// TwinCAT 3 PLC project Test
// ProgramVersion: 3.1.4026.24
// libraries:
//   Tc2_Standard, * (Beckhoff Automation GmbH)
//   Tc2_System, * (Beckhoff Automation GmbH)
// project tree:
//   DUTs/AMR/ stJoint2.TcDUT, stPose2D.TcDUT, stTarget2D.TcDUT
//   DUTs/BaseActions/ ITF_BA_6Axis.TcIO, ITF_BA_AMR.TcIO, ITF_BA_Scara.TcIO
//   DUTs/BasicRobot/ eMode.TcDUT, stFrame.TcDUT, stPose.TcDUT, stTarget.TcDUT
//   DUTs/Communication/ eCommunicationState.TcDUT, ITF_CommunicationModul_1.TcIO, ST_CommunicationConfig_1.TcDUT
//   DUTs/DB/ ST_Robot.TcDUT, ST_SQLValue.TcDUT
//   DUTs/Error/ eSeverity.TcDUT, stError.TcDUT
//   DUTs/ ITF_0_BaseComponent.TcIO, ITF_1_Robot.TcIO, ITF_1_Skill.TcIO, ITF_2_6AxisRobot.TcIO, ITF_2_AMR.TcIO, ITF_CommunicationModul.TcIO, ITF_Tool.TcIO, ST_CommunicationConfig.TcDUT
//   DUTs/Manipulator/ ITF_Tool_1.TcIO, stJoint6.TcDUT, stPose3D.TcDUT, stTarget3D.TcDUT
//   DUTs/StateMachine/ eInternalTransitions.TcDUT, eResult.TcDUT, eState.TcDUT, eSupervisoryTransitions.TcDUT
//   GVLs/ OPCUA.TcGVL, SKILLS.TcGVL
//   / PlcTask.TcTTO
//   POUs/Archiv/ FB_Axis.TcPOU
//   POUs/ FB_Base.TcPOU, FB_Helper.TcPOU, FB_PickPlaceSkill.TcPOU, FB_PostgreSQLClient.TcPOU, FB_ROB.TcPOU, FB_ROB_AMR.TcPOU, FB_ROB_MANIP.TcPOU, FB_Skill.TcPOU, FB_SkillHandler.TcPOU, FB_Tool.TcPOU, FB_UR5.TcPOU, MAIN_1.TcPOU, Test.TcPOU
//   POUs/Robots/ FB_OmronLD90.TcPOU, FB_ROB_1.TcPOU, FB_ROB_AMR_1.TcPOU, FB_ROB_MANIP_1.TcPOU, FB_UR5_1.TcPOU
//   POUs/Skills/ FB_SkillHandler_1.TcPOU, FB_Skill_1.TcPOU, Skill_LoadDeliverReturn.TcPOU, Skill_PickPlace.TcPOU

CONFIGURATION Test
    RESOURCE PLC ON TwinCAT3
        TASK PlcTask(INTERVAL := T#10ms, PRIORITY := 21);
        PROGRAM MAIN WITH PlcTask : MAIN;
    END_RESOURCE
END_CONFIGURATION

// ---- DUTs/AMR/stJoint2.TcDUT
TYPE stJoint2 :
STRUCT
	left : LREAL;
	right : LREAL;
END_STRUCT
END_TYPE

// ---- DUTs/AMR/stPose2D.TcDUT
TYPE stPose2D EXTENDS stPose :
STRUCT
	theta : LREAL;
END_STRUCT
END_TYPE

// ---- DUTs/AMR/stTarget2D.TcDUT
TYPE stTarget2D EXTENDS stTarget :
STRUCT
	pose : stPose2D;
END_STRUCT
END_TYPE

// ---- DUTs/BasicRobot/eMode.TcDUT
{attribute 'qualified_only'}
{attribute 'strict'}
TYPE eMode :
(
	Manual := 0,
	Automatic := 1
);
END_TYPE

// ---- DUTs/BasicRobot/stFrame.TcDUT
TYPE stFrame :
STRUCT
	frameId: UINT;
END_STRUCT
END_TYPE

// ---- DUTs/BasicRobot/stPose.TcDUT
TYPE stPose :
STRUCT
	x : LREAL;
	y : LREAL;
END_STRUCT
END_TYPE

// ---- DUTs/BasicRobot/stTarget.TcDUT
TYPE stTarget :
STRUCT
	name : STRING(80);
	frameId : INT;
END_STRUCT
END_TYPE

// ---- DUTs/Communication/eCommunicationState.TcDUT
{attribute 'qualified_only'}
{attribute 'strict'}
{attribute 'to_string'}
TYPE eCommunicationState :
(
	DISCONNECTED,
    CONNECTING,
    CONNECTED,
    DISCONNECTING,
    ERROR
);
END_TYPE

// ---- DUTs/Communication/ST_CommunicationConfig_1.TcDUT
TYPE ST_CommunicationConfig_1 :
STRUCT

    sIpAddress : STRING(15) := '192.168.0.10';
    nPort : UINT := 7171;
	sUsername: STRING(128):= '';
    sPassword : STRING(128) := '';
    tTimeout : TIME := T#5S;
    bAutoReconnect : BOOL := TRUE;
END_STRUCT
END_TYPE

// ---- DUTs/DB/ST_Robot.TcDUT
TYPE ST_Robot :
STRUCT
    id           : DINT;
    name         : STRING(80);
    manufacturer : STRING(80);
    model        : STRING(80);
    robot_type   : STRING(80);
    axes         : DINT;
    payload      : LREAL;
    reach        : LREAL;
    controller   : STRING(80);
    ip_address   : STRING(40);
END_STRUCT
END_TYPE

// ---- DUTs/DB/ST_SQLValue.TcDUT
TYPE ST_SQLValue  :
STRUCT
    sValue : STRING(255);
END_STRUCT
END_TYPE

// ---- DUTs/Error/eSeverity.TcDUT
{attribute 'qualified_only'}
{attribute 'strict'}
TYPE eSeverity :
(
	Info := 0,
	Warning := 1,
	Error := 2,
	Critical := 3
);
END_TYPE

// ---- DUTs/Error/stError.TcDUT
TYPE stError :
STRUCT
	code : INT;
	message : STRING(255);
	timestamp : DATE_AND_TIME;
	severity : eSeverity;
END_STRUCT
END_TYPE

// ---- DUTs/Manipulator/stJoint6.TcDUT
TYPE stJoint6 :
STRUCT
	joint1 : LREAL;
	joint2 : LREAL;
	joint3 : LREAL;
	joint4 : LREAL;
	joint5 : LREAL;
	joint6 : LREAL;
END_STRUCT
END_TYPE

// ---- DUTs/Manipulator/stPose3D.TcDUT
TYPE stPose3D EXTENDS stPose :
STRUCT
	z : LREAL;
	rx : LREAL;
	ry : LREAL;
	rz : LREAL;
END_STRUCT
END_TYPE

// ---- DUTs/Manipulator/stTarget3D.TcDUT
TYPE stTarget3D EXTENDS stTarget :
STRUCT
	pose : stPose3D;
END_STRUCT
END_TYPE

// ---- DUTs/StateMachine/eInternalTransitions.TcDUT
{attribute 'qualified_only'}
{attribute 'strict'}
TYPE eInternalTransitions :
(
	Configuring := 0,
	CleaningUp := 1,
	ShuttingDown := 2,
	Activating := 3,
	Deactivating := 4,
	ErrorProcessing := 5
);
END_TYPE

// ---- DUTs/StateMachine/eResult.TcDUT
{attribute 'qualified_only'}
{attribute 'strict'}
{attribute 'to_string'}
TYPE eResult :
(
	NONE := 0,
	SUCCESS := 1,
	FAILURE := 2,
	ERROR	:= 3
);
END_TYPE

// ---- DUTs/StateMachine/eState.TcDUT
{attribute 'qualified_only'}
{attribute 'strict'}
TYPE eState :
(
	None 			:= 0,
	Unconfigured 	:= 1,
	Inactive 		:= 2,
	Active 			:= 3,
	Finalized 		:= 4,
	Configuring		:= 5,
	CleaningUp 		:= 6,
	Activating 		:= 7,
	Deactivating 	:= 8,
	ShuttingDown 	:= 9,
	ErrorProcessing := 10
);
END_TYPE

// ---- DUTs/StateMachine/eSupervisoryTransitions.TcDUT
{attribute 'qualified_only'}
{attribute 'strict'}
TYPE eSupervisoryTransitions :
(
	create := 0,
	configure := 1,
	cleanup := 2,
	activate := 3,
	deactivate := 4,
	shutdown := 5,
	destroy := 6
);
END_TYPE

// ---- DUTs/ST_CommunicationConfig.TcDUT
TYPE ST_CommunicationConfig :
STRUCT
	sIPAdress: STRING;
	Port: UINT;
	
END_STRUCT
END_TYPE

// ---- GVLs/OPCUA.TcGVL
{attribute 'qualified_only'}
VAR_GLOBAL
	{attribute 'OPC.UA.DA.StructuredType' := '1'}
	{attribute 'OPC.UA.DA' := '1'}
	ROB : ARRAY[1..3] of FB_ROB;
END_VAR

// ---- GVLs/SKILLS.TcGVL
{attribute 'qualified_only'}
VAR_GLOBAL
	PnP: FB_PickPlaceSkill;
END_VAR

// ---- DUTs/BaseActions/ITF_BA_6Axis.TcIO
INTERFACE ITF_BA_6Axis

METHOD MC_ChangeSpeedOverride : INT
VAR_INPUT
	factor: REAL;
END_VAR
END_METHOD

METHOD MC_MoveAxesAbsolute : BOOL
VAR_INPUT
	target: stTarget3D;
END_VAR
END_METHOD

METHOD MC_MoveAxesRelative : BOOL
VAR_INPUT
	axes: ARRAY[1..6] OF FB_Axis;
	offsets: ARRAY[1..6] OF REAL;
END_VAR
END_METHOD

METHOD MC_MoveLinearAbsolute : BOOL
VAR_INPUT
	target: stTarget3D;
END_VAR
END_METHOD

METHOD PUBLIC MC_ReadAnalogInput : LREAL
VAR_INPUT
	input : INT;
END_VAR
END_METHOD

METHOD PUBLIC MC_ReadDigitalInput : BOOL
VAR_INPUT
	input : INT;
END_VAR
END_METHOD

METHOD PUBLIC MC_SetDigitalOutput : BOOL
VAR_INPUT
	output : INT;
	value : BOOL;
END_VAR
END_METHOD

METHOD PUBLIC MC_SetOperationMode : BOOL
VAR_INPUT
	mode: eMode;
END_VAR
END_METHOD

END_INTERFACE

// ---- DUTs/BaseActions/ITF_BA_AMR.TcIO
INTERFACE ITF_BA_AMR

METHOD MC_ChangeSpeedOverride : INT
VAR_INPUT
	factor: REAL;
END_VAR
END_METHOD

METHOD MC_MoveAxesAbsolute : BOOL
VAR_INPUT
	target: stTarget3D;
END_VAR
END_METHOD

METHOD MC_MoveAxesRelative : BOOL
VAR_INPUT
	axes: ARRAY[1..6] OF FB_Axis;
	offsets: ARRAY[1..6] OF REAL;
END_VAR
END_METHOD

METHOD MC_MoveLinearAbsolute : BOOL
VAR_INPUT
	target: stTarget3D;
END_VAR
END_METHOD

METHOD PUBLIC MC_ReadAnalogInput : LREAL
VAR_INPUT
	input : INT;
END_VAR
END_METHOD

METHOD PUBLIC MC_ReadDigitalInput : BOOL
VAR_INPUT
	input : INT;
END_VAR
END_METHOD

METHOD PUBLIC MC_SetDigitalOutput : BOOL
VAR_INPUT
	output : INT;
	value : BOOL;
END_VAR
END_METHOD

METHOD PUBLIC MC_SetOperationMode : BOOL
VAR_INPUT
	mode: eMode;
END_VAR
END_METHOD

END_INTERFACE

// ---- DUTs/BaseActions/ITF_BA_Scara.TcIO
INTERFACE ITF_BA_Scara

METHOD MC_ChangeSpeedOverride : INT
VAR_INPUT
	factor: REAL;
END_VAR
END_METHOD

METHOD MC_MoveAxesAbsolute : BOOL
VAR_INPUT
	target: stTarget3D;
END_VAR
END_METHOD

METHOD MC_MoveAxesRelative : BOOL
VAR_INPUT
	axes: ARRAY[1..6] OF FB_Axis;
	offsets: ARRAY[1..6] OF REAL;
END_VAR
END_METHOD

METHOD MC_MoveLinearAbsolute : BOOL
VAR_INPUT
	target: stTarget3D;
END_VAR
END_METHOD

METHOD PUBLIC MC_ReadAnalogInput : LREAL
VAR_INPUT
	input : INT;
END_VAR
END_METHOD

METHOD PUBLIC MC_ReadDigitalInput : BOOL
VAR_INPUT
	input : INT;
END_VAR
END_METHOD

METHOD PUBLIC MC_SetDigitalOutput : BOOL
VAR_INPUT
	output : INT;
	value : BOOL;
END_VAR
END_METHOD

METHOD PUBLIC MC_SetOperationMode : BOOL
VAR_INPUT
	mode: eMode;
END_VAR
END_METHOD

END_INTERFACE

// ---- DUTs/Communication/ITF_CommunicationModul_1.TcIO
INTERFACE ITF_CommunicationModul_1

METHOD Connect : BOOL
VAR_INPUT
END_VAR
END_METHOD

PROPERTY Connected : BOOL
GET
END_GET
END_PROPERTY

METHOD Disconnect : BOOL
VAR_INPUT
END_VAR
END_METHOD

METHOD ResetConnection : BOOL
VAR_INPUT
END_VAR
END_METHOD

END_INTERFACE

// ---- DUTs/ITF_0_BaseComponent.TcIO
INTERFACE ITF_0_BaseComponent

METHOD M_activate : BOOL
VAR_INPUT
END_VAR
END_METHOD

METHOD M_cleanup : BOOL
VAR_INPUT
END_VAR
END_METHOD

METHOD M_configure : BOOL
VAR_INPUT
END_VAR
END_METHOD

METHOD M_deactivate : BOOL
VAR_INPUT
END_VAR
END_METHOD

METHOD M_destroy : BOOL
VAR_INPUT
END_VAR
END_METHOD

METHOD M_shutdown : BOOL
VAR_INPUT
END_VAR
END_METHOD

METHOD onActivate : BOOL
VAR_INPUT
END_VAR
END_METHOD

METHOD onCleanup : BOOL
VAR_INPUT
END_VAR
END_METHOD

METHOD onConfigure : BOOL
VAR_INPUT
END_VAR
END_METHOD

METHOD onDeactivate : BOOL
VAR_INPUT
END_VAR
END_METHOD

METHOD onError : BOOL
VAR_INPUT
END_VAR
END_METHOD

METHOD onShutdown : BOOL
VAR_INPUT
END_VAR
END_METHOD

PROPERTY P_ID : UINT
GET
END_GET
SET
END_SET
END_PROPERTY

PROPERTY P_Name : String
GET
END_GET
END_PROPERTY

PROPERTY P_Path : String
GET
END_GET
END_PROPERTY

PROPERTY ABSTRACT P_State : eState
GET
END_GET
SET
END_SET
END_PROPERTY

END_INTERFACE

// ---- DUTs/ITF_1_Robot.TcIO
INTERFACE ITF_1_Robot EXTENDS ITF_0_BaseComponent

METHOD M_AUTO : BOOL
VAR_INPUT
END_VAR
END_METHOD

METHOD M_Disable : BOOL
VAR_INPUT
END_VAR
END_METHOD

METHOD M_DisableVelocityOverride : BOOL
VAR_INPUT
END_VAR
END_METHOD

METHOD M_Enable : BOOL
VAR_INPUT
END_VAR
END_METHOD

METHOD M_EnableVelocityOverride : BOOL
VAR_INPUT
END_VAR
END_METHOD

METHOD M_EStop : BOOL
VAR_INPUT
END_VAR
END_METHOD

METHOD M_MAN : BOOL
VAR_INPUT
END_VAR
END_METHOD

PROPERTY P_isInCollision : BOOL
GET
END_GET
END_PROPERTY

{warning 'Eigenschaftenimplementierung hinzufügen'}
PROPERTY P_JogSpeed : LREAL
GET
END_GET
SET
END_SET
END_PROPERTY

{warning 'Eigenschaftenimplementierung hinzufügen'}
PROPERTY P_RobotIsMoving : BOOL
GET
END_GET
END_PROPERTY

{warning 'Eigenschaftenimplementierung hinzufügen'}
PROPERTY P_RobotIsReady : BOOL
GET
END_GET
END_PROPERTY

END_INTERFACE

// ---- DUTs/ITF_1_Skill.TcIO
INTERFACE ITF_1_Skill EXTENDS ITF_0_BaseComponent

METHOD M_Pause : BOOL
VAR_INPUT
END_VAR
END_METHOD

METHOD M_Restart : BOOL
VAR_INPUT
END_VAR
END_METHOD

METHOD M_Resume : BOOL
VAR_INPUT
END_VAR
END_METHOD

METHOD M_Start : BOOL
VAR_INPUT
END_VAR
END_METHOD

METHOD M_Stop : BOOL
VAR_INPUT
END_VAR
END_METHOD

PROPERTY P_Busy : BOOL
GET
END_GET
END_PROPERTY

PROPERTY P_Done : BOOL
GET
END_GET
END_PROPERTY

END_INTERFACE

// ---- DUTs/ITF_2_6AxisRobot.TcIO
INTERFACE ITF_2_6AxisRobot IMPLEMENTS ITF_1_Robot

METHOD M_Home : BOOL
VAR_INPUT
END_VAR
END_METHOD

METHOD M_SwitchTool : UINT
VAR_INPUT
	tool: FB_Tool;
END_VAR
END_METHOD

{warning 'Eigenschaftenimplementierung hinzufügen'}
PROPERTY P_ActualAxisPos :stJoint6
GET
END_GET
END_PROPERTY

PROPERTY P_ActualJointVelocity : stJoint6
GET
END_GET
END_PROPERTY

{warning 'Eigenschaftenimplementierung hinzufügen'}
PROPERTY P_ActualTCPPos :stPose3D
GET
END_GET
END_PROPERTY

PROPERTY P_ActualTCPVelocity : stPose3D
GET
END_GET
END_PROPERTY

PROPERTY P_CurrentFrame : stFrame
GET
END_GET
SET
END_SET
END_PROPERTY

PROPERTY P_CurrentFrameID : UINT
GET
END_GET
END_PROPERTY

PROPERTY P_CurrentTool : FB_Tool
GET
END_GET
SET
END_SET
END_PROPERTY

PROPERTY P_IsInHomePosition : BOOL
GET
END_GET
END_PROPERTY

{warning 'Add property implementation'}
PROPERTY P_TargetReached : BOOL
GET
END_GET
END_PROPERTY

END_INTERFACE

// ---- DUTs/ITF_2_AMR.TcIO
INTERFACE ITF_2_AMR IMPLEMENTS ITF_1_Robot

METHOD M_Dock : BOOL
VAR_INPUT
END_VAR
END_METHOD

PROPERTY P_ActualAxisPos :stJoint2
GET
END_GET
END_PROPERTY

PROPERTY P_ActualJointVelocity : stJoint2
GET
END_GET
END_PROPERTY

PROPERTY P_ActualTCPPos :stPose2D
GET
END_GET
END_PROPERTY

PROPERTY P_ActualTCPVelocity : stPose2D
GET
END_GET
END_PROPERTY

PROPERTY P_IsDocked : BOOL
GET
END_GET
END_PROPERTY

{warning 'Add property implementation'}
PROPERTY P_TargetReached : BOOL
GET
END_GET
END_PROPERTY

END_INTERFACE

// ---- DUTs/ITF_CommunicationModul.TcIO
INTERFACE ITF_CommunicationModul

METHOD M_Connect : BOOL
VAR_INPUT
END_VAR
END_METHOD

METHOD M_Disconnect : BOOL
VAR_INPUT
END_VAR
END_METHOD

METHOD M_ResetConnection : BOOL
VAR_INPUT
END_VAR
END_METHOD

PROPERTY P_bConnected : BOOL
GET
END_GET
END_PROPERTY

END_INTERFACE

// ---- DUTs/ITF_Tool.TcIO
INTERFACE ITF_Tool

METHOD Grip : BOOL
VAR_INPUT
END_VAR
END_METHOD

METHOD Release : BOOL
VAR_INPUT
END_VAR
END_METHOD

END_INTERFACE

// ---- DUTs/Manipulator/ITF_Tool_1.TcIO
INTERFACE ITF_Tool_1

METHOD Grip : BOOL
VAR_INPUT
END_VAR
END_METHOD

METHOD Release : BOOL
VAR_INPUT
END_VAR
END_METHOD

END_INTERFACE

// ---- POUs/FB_ROB.TcPOU
FUNCTION_BLOCK FB_ROB EXTENDS FB_Base IMPLEMENTS ITF_1_Robot

// VAR_IN_OUT
// 	Skills: ARRAY[1..3] OF FB_Skill;
// END_VAR
VAR_INPUT
	ComConfig: ST_CommunicationConfig;
END_VAR


VAR_OUTPUT
	_inCollision: BOOL;
END_VAR
VAR
	_enabled: BOOL;
	_mode: eMode;
	_locked: BOOL;
	
	velovr: BOOL;
	velfact: REAL;
	
	DBClient: FB_PostgreSQLClient;
	

END_VAR

//State Machine

DBClient();

{warning 'Add method implementation '}
METHOD M_AUTO : BOOL
_mode:=eMode.Automatic;
END_METHOD

{warning 'Add method implementation '}
METHOD M_Disable : BOOL
_enabled:=FALSE;
M_deactivate();
END_METHOD

{warning 'Add method implementation '}
METHOD M_DisableVelocityOverride : BOOL
velovr:=False;
END_METHOD

{warning 'Add method implementation '}
METHOD M_Enable : BOOL
_enabled:=TRUE;
END_METHOD

{warning 'Add method implementation '}
METHOD M_EnableVelocityOverride : BOOL
velovr:=True;
END_METHOD

{warning 'Add method implementation '}
METHOD M_EStop : BOOL
END_METHOD

{warning 'Add method implementation '}
METHOD M_MAN : BOOL
_mode:=eMode.Manual;
END_METHOD

{warning 'Add method implementation '}
METHOD MC_ChangeSpeedOverride : INT
VAR_INPUT
	factor	: REAL;
END_VAR
velfact:=factor;
END_METHOD

METHOD onActivate : BOOL
// ---- Init ----
transitionresult:=eResult.None;



// ---- Change ----

// _mode:= eMode.Automatic;




// ---- Check ----
transitionresult := eResult.SUCCESS;


// ---- Change State ----
IF transitionresult= eResult.SUCCESS THEN
	P_State:=eState.Active;
ELSIF transitionresult= eResult.FAILURE THEN
	P_State:=eState.Inactive;
ELSIF transitionresult= eResult.ERROR THEN
	P_State:=eState.ErrorProcessing;
ELSE
	ADSLOGSTR(ADSLOG_MSGTYPE_WARN,'Transitionresult from onActivate is None','');
END_IF
END_METHOD

METHOD onCleanup : BOOL
// ---- Init ----
transitionresult:=eResult.None;



// ---- Change ----

_mode:= eMode.Manual;




// ---- Check ----
transitionresult := eResult.SUCCESS;


// ---- Change State ----
IF transitionresult= eResult.SUCCESS THEN
	P_State:=eState.Unconfigured;
ELSIF transitionresult= eResult.FAILURE THEN
	ADSLOGSTR(ADSLOG_MSGTYPE_WARN,'Transitionresult from onCleanup is FAILURE ','');
ELSIF transitionresult= eResult.ERROR THEN
	P_State:=eState.ErrorProcessing;
ELSE
	ADSLOGSTR(ADSLOG_MSGTYPE_WARN,'Transitionresult from onCleanup is NONE','');
END_IF
END_METHOD

METHOD onConfigure : BOOL
// ---- Init ----
transitionresult:=eResult.None;



// ---- Change ----

_mode:= eMode.Manual;




// ---- Check ----
transitionresult := eResult.SUCCESS;


// ---- Change State ----
IF transitionresult= eResult.SUCCESS THEN
	P_State:=eState.Inactive;
ELSIF transitionresult= eResult.FAILURE THEN
	P_State:=eState.Unconfigured;
ELSIF transitionresult= eResult.ERROR THEN
	P_State:=eState.ErrorProcessing;
ELSE
	ADSLOGSTR(ADSLOG_MSGTYPE_WARN,'Transitionresult from onConfigure is None','');
END_IF
END_METHOD

METHOD onDeactivate : BOOL
// ---- Init ----
transitionresult:=eResult.None;



// ---- Change ----

_mode:= eMode.Manual;




// ---- Check ----
transitionresult := eResult.SUCCESS;


// ---- Change State ----
IF transitionresult= eResult.SUCCESS THEN
	P_State:=eState.Inactive;
ELSIF transitionresult= eResult.FAILURE THEN
	ADSLOGSTR(ADSLOG_MSGTYPE_WARN,'Transitionresult from onDeactivate is FAILURE','');
ELSIF transitionresult= eResult.ERROR THEN
	P_State:=eState.ErrorProcessing;
ELSE
	ADSLOGSTR(ADSLOG_MSGTYPE_WARN,'Transitionresult from onDeactivate is None','');
END_IF
END_METHOD

METHOD onError : BOOL
// ---- Init ----
transitionresult:=eResult.None;



// ---- Change ----

_mode:= eMode.Manual;




// ---- Check ----
transitionresult := eResult.SUCCESS;


// ---- Change State ----
IF transitionresult= eResult.SUCCESS THEN
	P_State:=eState.Unconfigured;
ELSIF transitionresult= eResult.FAILURE THEN
	P_State:=eState.Finalized;
ELSIF transitionresult= eResult.ERROR THEN
	ADSLOGSTR(ADSLOG_MSGTYPE_WARN,'Transitionresult from onError is Error','');
ELSE
	ADSLOGSTR(ADSLOG_MSGTYPE_WARN,'Transitionresult from onError is None','');
END_IF
END_METHOD

METHOD onShutdown : BOOL
// ---- Init ----
transitionresult:=eResult.None;



// ---- Change ----

_mode:= eMode.Manual;




// ---- Check ----
transitionresult := eResult.SUCCESS;


// ---- Change State ----
IF transitionresult= eResult.SUCCESS THEN
	P_State:=eState.Finalized;
ELSIF transitionresult= eResult.FAILURE THEN
	ADSLOGSTR(ADSLOG_MSGTYPE_WARN,'Transitionresult from onShutdown is FAILURE','');
ELSIF transitionresult= eResult.ERROR THEN
	P_State:=eState.ErrorProcessing;
ELSE
	ADSLOGSTR(ADSLOG_MSGTYPE_WARN,'Transitionresult from onShutdown is None','');
END_IF
END_METHOD

{warning 'Add property implementation'}
PROPERTY P_isInCollision : BOOL
GET
P_isInCollision:=_inCollision;
END_GET
END_PROPERTY

{warning 'Add property implementation'}
PROPERTY P_JogSpeed : LREAL
GET
END_GET
SET
END_SET
END_PROPERTY

{warning 'Add property implementation'}
PROPERTY P_RobotIsMoving : BOOL
GET
END_GET
END_PROPERTY

{warning 'Add property implementation'}
PROPERTY P_RobotIsReady : BOOL
GET
END_GET
END_PROPERTY

END_FUNCTION_BLOCK

// ---- POUs/FB_Base.TcPOU
{attribute 'reflection'} 
FUNCTION_BLOCK ABSTRACT FB_Base EXTENDS  FB_SkillHandler  IMPLEMENTS ITF_0_BaseComponent
VAR_INPUT
END_VAR
VAR_OUTPUT
END_VAR
VAR
	{attribute 'instance-path'} 
    {attribute 'noinit'} 
    sPath : STRING; 
	{attribute 'instance-name'}
	{attribute 'noinit'} 
	sInstanceName: STRING;
	_autoboot: BOOL:=TRUE;		//If True, StateMachine trys automatic to reach State "ACTIV" otherwise each transition must be called manually
	
	transitionresult: eResult;
	_state: eState :=eState.Unconfigured;
	

	dummy: INT;
END_VAR

StateMachine();

{warning 'Add method implementation '}
METHOD M_activate : BOOL
IF P_State=eState.Inactive THEN
	P_State:=eState.Activating;
END_IF
END_METHOD

{warning 'Add method implementation '}
METHOD M_cleanup : BOOL
IF P_State=eState.Inactive THEN
	P_State:=eState.CleaningUp;
END_IF
END_METHOD

{warning 'Add method implementation '}
METHOD M_configure : BOOL
IF P_State=eState.Unconfigured THEN
	P_State:=eState.Configuring;
END_IF
END_METHOD

{warning 'Add method implementation '}
METHOD M_deactivate : BOOL
IF P_State=eState.Active THEN
	P_State:=eState.Deactivating;
END_IF
END_METHOD

{warning 'Add method implementation '}
METHOD M_destroy : BOOL
IF P_State=eState.Finalized THEN
	P_State:=eState.Unconfigured;
END_IF
END_METHOD

{warning 'Add method implementation '}
METHOD M_shutdown : BOOL
IF P_State=eState.Inactive OR P_State=eState.Unconfigured OR P_State=eState.Active THEN
	P_State:=eState.ShuttingDown;
END_IF
END_METHOD

METHOD onActivate : BOOL
// ---- Init ----
transitionresult:=eResult.None;



// ---- Change ----



// ---- Check ----
transitionresult := eResult.SUCCESS;


// ---- Change State ----
IF transitionresult= eResult.SUCCESS THEN
	P_State:=eState.Active;
ELSIF transitionresult= eResult.FAILURE THEN
	P_State:=eState.Inactive;
ELSIF transitionresult= eResult.ERROR THEN
	P_State:=eState.ErrorProcessing;
ELSE
	ADSLOGSTR(ADSLOG_MSGTYPE_WARN,'Transitionresult from onActivate is None','');
END_IF
END_METHOD

METHOD onCleanup : BOOL
// ---- Init ----
transitionresult:=eResult.None;



// ---- Change ----



// ---- Check ----
transitionresult := eResult.SUCCESS;


// ---- Change State ----
IF transitionresult= eResult.SUCCESS THEN
	P_State:=eState.Unconfigured;
ELSIF transitionresult= eResult.FAILURE THEN
	ADSLOGSTR(ADSLOG_MSGTYPE_WARN,'Transitionresult from onCleanup is FAILURE ','');
ELSIF transitionresult= eResult.ERROR THEN
	P_State:=eState.ErrorProcessing;
ELSE
	ADSLOGSTR(ADSLOG_MSGTYPE_WARN,'Transitionresult from onCleanup is NONE','');
END_IF
END_METHOD

METHOD onConfigure : BOOL
// ---- Init ----
transitionresult:=eResult.None;



// ---- Change ----




// ---- Check ----
transitionresult := eResult.SUCCESS;


// ---- Change State ----
IF transitionresult= eResult.SUCCESS THEN
	P_State:=eState.Inactive;
ELSIF transitionresult= eResult.FAILURE THEN
	P_State:=eState.Unconfigured;
ELSIF transitionresult= eResult.ERROR THEN
	P_State:=eState.ErrorProcessing;
ELSE
	ADSLOGSTR(ADSLOG_MSGTYPE_WARN,'Transitionresult from onConfigure is None','');
END_IF
END_METHOD

METHOD onDeactivate : BOOL
// ---- Init ----
transitionresult:=eResult.None;



// ---- Change ----



// ---- Check ----
transitionresult := eResult.SUCCESS;


// ---- Change State ----
IF transitionresult= eResult.SUCCESS THEN
	P_State:=eState.Inactive;
ELSIF transitionresult= eResult.FAILURE THEN
	ADSLOGSTR(ADSLOG_MSGTYPE_WARN,'Transitionresult from onDeactivate is FAILURE','');
ELSIF transitionresult= eResult.ERROR THEN
	P_State:=eState.ErrorProcessing;
ELSE
	ADSLOGSTR(ADSLOG_MSGTYPE_WARN,'Transitionresult from onDeactivate is None','');
END_IF
END_METHOD

METHOD onError : BOOL
// ---- Init ----
transitionresult:=eResult.None;



// ---- Change ----




// ---- Check ----
transitionresult := eResult.SUCCESS;


// ---- Change State ----
IF transitionresult= eResult.SUCCESS THEN
	P_State:=eState.Unconfigured;
ELSIF transitionresult= eResult.FAILURE THEN
	P_State:=eState.Finalized;
ELSIF transitionresult= eResult.ERROR THEN
	ADSLOGSTR(ADSLOG_MSGTYPE_WARN,'Transitionresult from onError is Error','');
ELSE
	ADSLOGSTR(ADSLOG_MSGTYPE_WARN,'Transitionresult from onError is None','');
END_IF
END_METHOD

METHOD onShutdown : BOOL
// ---- Init ----
transitionresult:=eResult.None;



// ---- Change ----



// ---- Check ----
transitionresult := eResult.SUCCESS;


// ---- Change State ----
IF transitionresult= eResult.SUCCESS THEN
	P_State:=eState.Finalized;
ELSIF transitionresult= eResult.FAILURE THEN
	ADSLOGSTR(ADSLOG_MSGTYPE_WARN,'Transitionresult from onShutdown is FAILURE','');
ELSIF transitionresult= eResult.ERROR THEN
	P_State:=eState.ErrorProcessing;
ELSE
	ADSLOGSTR(ADSLOG_MSGTYPE_WARN,'Transitionresult from onShutdown is None','');
END_IF
END_METHOD

PROPERTY P_AutoBoot : BOOL
GET
P_AutoBoot:=_autoboot;
END_GET
SET
_autoboot:=P_AutoBoot;
END_SET
END_PROPERTY

{warning 'Add property implementation'}
PROPERTY P_ID : UINT
GET
END_GET
SET
END_SET
END_PROPERTY

{warning 'Add property implementation'}
PROPERTY P_Name : STRING
GET


P_Name:=sInstanceName;
END_GET
END_PROPERTY

{warning 'Add property implementation'}
PROPERTY P_Path : STRING
GET
P_Path:=sPath;
END_GET
END_PROPERTY

{warning 'Add property implementation'}
PROPERTY P_State : eState
GET
P_State:=_state;
END_GET
SET
_state:=P_State;
END_SET
END_PROPERTY

METHOD StateMachine : eState
VAR_INPUT
END_VAR
CASE _state OF
	eState.Unconfigured:
		IF _autoboot THEN
			M_configure();
		END_IF
	eState.Inactive:		//IDLE
// 		IF _autoboot THEN
// 			M_activate();
// 		END_IF
	eState.Active:
		dummy:=1;
	eState.Finalized:
		M_destroy();
	
	
	//Transitions States
	eState.Configuring:
		onConfigure();
	eState.Activating:
		onActivate();
	eState.Deactivating:
		onDeactivate();
	eState.ErrorProcessing:
		onError();
	eState.CleaningUp:
		onCleanup();
	eState.ShuttingDown:
		onShutdown();
		
END_CASE
END_METHOD

END_FUNCTION_BLOCK

// ---- POUs/FB_SkillHandler.TcPOU
FUNCTION_BLOCK FB_SkillHandler
VAR_INPUT
END_VAR
VAR_OUTPUT
END_VAR
VAR
	activSkill: POINTER TO FB_SKILL;
	_finished: BOOL;
END_VAR

IF activSkill^.bDone THEN
	_finished:=True;
END_IF

METHOD AbortActifSkill : BOOL
VAR_INPUT
END_VAR
activSkill^.M_Stop();
END_METHOD

METHOD CallSkill : BOOL
VAR_INPUT
	pSkill : POINTER TO FB_SKILL;
END_VAR
activSkill:= pSkill;

//TODO Checks

pSkill^.M_Start();
END_METHOD

PROPERTY P_ActiveSkillFinished : BOOL
GET
P_ActiveSkillFinished := _finished;
END_GET
END_PROPERTY

PROPERTY P_GetActivSkill : POINTER TO FB_SKILL
GET
P_GetActivSkill := activSkill;
END_GET
END_PROPERTY

END_FUNCTION_BLOCK

// ---- POUs/FB_Skill.TcPOU
FUNCTION_BLOCK FB_Skill EXTENDS FB_Base IMPLEMENTS  ITF_1_Skill
VAR_INPUT
	SFCInit, SFCPause, SFCReset: BOOL;
END_VAR
VAR_OUTPUT
	bBusy, bDone: BOOL;
	SFCError: BOOL;
	SFCCurrentStep: STRING;
END_VAR
VAR
	SubSkillHandler : FB_SkillHandler;
END_VAR

{warning 'Add method implementation '}
METHOD M_Pause : BOOL
IF _state=eState.Active THEN
	SFCPause:=TRUE;
END_IF
END_METHOD

{warning 'Add method implementation '}
METHOD M_Restart : BOOL //Stay activ, but restart
SFCReset:=True;
END_METHOD

{warning 'Add method implementation '}
METHOD M_Resume : BOOL
SFCPause:=False;
END_METHOD

{warning 'Add method implementation '}
METHOD M_Start : BOOL
M_activate();
END_METHOD

{warning 'Add method implementation '}
METHOD M_Stop : BOOL
IF _state=eState.Active THEN
	SFCPause:=TRUE;
	M_deactivate();
END_IF
END_METHOD

METHOD onActivate : BOOL
// ---- Init ----
transitionresult:=eResult.None;



// ---- Change ----




// ---- Check ----
transitionresult := eResult.SUCCESS;


// ---- Change State ----
IF transitionresult= eResult.SUCCESS THEN
	P_State:=eState.Active;
ELSIF transitionresult= eResult.FAILURE THEN
	P_State:=eState.Inactive;
ELSIF transitionresult= eResult.ERROR THEN
	P_State:=eState.ErrorProcessing;
ELSE
	ADSLOGSTR(ADSLOG_MSGTYPE_WARN,'Transitionresult from onActivate is None','');
END_IF
END_METHOD

METHOD onCleanup : BOOL
// ---- Init ----
transitionresult:=eResult.None;



// ---- Change ----



// ---- Check ----
transitionresult := eResult.SUCCESS;


// ---- Change State ----
IF transitionresult= eResult.SUCCESS THEN
	P_State:=eState.Unconfigured;
ELSIF transitionresult= eResult.FAILURE THEN
	ADSLOGSTR(ADSLOG_MSGTYPE_WARN,'Transitionresult from onCleanup is FAILURE ','');
ELSIF transitionresult= eResult.ERROR THEN
	P_State:=eState.ErrorProcessing;
ELSE
	ADSLOGSTR(ADSLOG_MSGTYPE_WARN,'Transitionresult from onCleanup is NONE','');
END_IF
END_METHOD

METHOD onConfigure : BOOL
// ---- Init ----
transitionresult:=eResult.None;



// ---- Change ----


// ---- Check ----
transitionresult := eResult.SUCCESS;


// ---- Change State ----
IF transitionresult= eResult.SUCCESS THEN
	P_State:=eState.Inactive;
ELSIF transitionresult= eResult.FAILURE THEN
	P_State:=eState.Unconfigured;
ELSIF transitionresult= eResult.ERROR THEN
	P_State:=eState.ErrorProcessing;
ELSE
	ADSLOGSTR(ADSLOG_MSGTYPE_WARN,'Transitionresult from onConfigure is None','');
END_IF
END_METHOD

METHOD onDeactivate : BOOL
// ---- Init ----
transitionresult:=eResult.None;



// ---- Change ----
 //Stopping SFC



// ---- Check ----
transitionresult := eResult.SUCCESS;


// ---- Change State ----
IF transitionresult= eResult.SUCCESS THEN
	P_State:=eState.Inactive;
ELSIF transitionresult= eResult.FAILURE THEN
	ADSLOGSTR(ADSLOG_MSGTYPE_WARN,'Transitionresult from onDeactivate is FAILURE','');
ELSIF transitionresult= eResult.ERROR THEN
	P_State:=eState.ErrorProcessing;
ELSE
	ADSLOGSTR(ADSLOG_MSGTYPE_WARN,'Transitionresult from onDeactivate is None','');
END_IF
END_METHOD

METHOD onError : BOOL
// ---- Init ----
transitionresult:=eResult.None;



// ---- Change ----





// ---- Check ----
transitionresult := eResult.SUCCESS;


// ---- Change State ----
IF transitionresult= eResult.SUCCESS THEN
	P_State:=eState.Unconfigured;
ELSIF transitionresult= eResult.FAILURE THEN
	P_State:=eState.Finalized;
ELSIF transitionresult= eResult.ERROR THEN
	ADSLOGSTR(ADSLOG_MSGTYPE_WARN,'Transitionresult from onError is Error','');
ELSE
	ADSLOGSTR(ADSLOG_MSGTYPE_WARN,'Transitionresult from onError is None','');
END_IF
END_METHOD

METHOD onShutdown : BOOL
// ---- Init ----
transitionresult:=eResult.None;



// ---- Change ----




// ---- Check ----
transitionresult := eResult.SUCCESS;


// ---- Change State ----
IF transitionresult= eResult.SUCCESS THEN
	P_State:=eState.Finalized;
ELSIF transitionresult= eResult.FAILURE THEN
	ADSLOGSTR(ADSLOG_MSGTYPE_WARN,'Transitionresult from onShutdown is FAILURE','');
ELSIF transitionresult= eResult.ERROR THEN
	P_State:=eState.ErrorProcessing;
ELSE
	ADSLOGSTR(ADSLOG_MSGTYPE_WARN,'Transitionresult from onShutdown is None','');
END_IF
END_METHOD

{warning 'Add property implementation'}
PROPERTY P_Busy : BOOL
GET
IF _state=eState.Active THEN
	P_Busy:=TRUE;
ELSE
	P_Busy:=FALSE;
END_IF
END_GET
END_PROPERTY

{warning 'Add property implementation'}
PROPERTY P_Done : BOOL
GET
P_Done:=bDone;
END_GET
END_PROPERTY

END_FUNCTION_BLOCK

// ---- POUs/FB_PostgreSQLClient.TcPOU
FUNCTION_BLOCK FB_PostgreSQLClient
VAR_INPUT
    bConnect : BOOL;
END_VAR

VAR_OUTPUT
    bConnected : BOOL;
    bError : BOOL;
    nErrorID : UDINT;
END_VAR

VAR
	sDBDatabase : STRING  := 'robotdata';
	sDBDriver : STRING  := 'PostgreSQL Unicode(x64)';
	sDBServer : STRING  := '192.168.250.102';
	nDBPort: UINT := 5432;
	sDBUserId : STRING := 'admin';
	sDBPassword : STRING  := '1';	


	bExecute: BOOL;
    fbDBOdbcAdd : FB_DBOdbcConnectionAdd;
    fbDBRecordSelect : FB_DBRecordSelect;

    hDBID : UDINT;

    bConnectExecute : BOOL;
    bQueryExecute : BOOL;

    sSQL : STRING(255);

    bInit : BOOL := TRUE;
	aa: BOOL;
END_VAR

VAR
	robot: ST_Robot;
END_VAR


IF NOT bConnected THEN
	Connect();
END_IF

IF aa THEN
	ReadRobots();
	aa:=False;
END_IF

METHOD Connect
IF NOT bConnected THEN

    bConnectExecute := TRUE;

    fbDBOdbcAdd(
        sDBDatabase := 'robotdata',
        sDBDriver := 'PostgreSQL Unicode(x64)',
        sDBServer := '192.168.250.102',
        nDBPort := 5432,
        sDBUserId := 'admin',
        sDBPassword := '1',
        hDBID => hDBID,
        bExecute := bConnectExecute
    );


    IF NOT fbDBOdbcAdd.bBusy THEN
        
        bConnectExecute := FALSE;

        IF fbDBOdbcAdd.bError THEN
            bError := TRUE;
            nErrorID := fbDBOdbcAdd.nErrID;
        ELSE
            bConnected := TRUE;
        END_IF

    END_IF

END_IF
END_METHOD

METHOD PUBLIC ExecuteSQL
VAR_INPUT
    sCommand : STRING;
END_VAR


IF bConnected THEN

    sSQL := sCommand;

    bQueryExecute := TRUE;


    fbDBRecordSelect(
			hDBID := hDBID,
			sSelectCmd := sCommand,
			pDestAddr := ADR(robot),
			cbRecordSize := SIZEOF(robot),
			nRecordIndex:=0,
			bExecute := bQueryExecute
		);


    IF NOT fbDBRecordSelect.bBusy THEN

        bQueryExecute := FALSE;

        IF fbDBRecordSelect.bError THEN
            bError := TRUE;
            nErrorID := fbDBRecordSelect.nErrID;
        END_IF

    END_IF

END_IF
END_METHOD

METHOD ReadRobots
VAR_INPUT
END_VAR
ExecuteSQL(
    sCommand := 'SELECT * FROM robots'
);
END_METHOD

END_FUNCTION_BLOCK

// ---- POUs/FB_PickPlaceSkill.TcPOU
FUNCTION_BLOCK FB_PickPlaceSkill EXTENDS FB_Skill
VAR_INPUT
	Rob: POINTER TO FB_ROB_MANIP;
	sPickReference: STRING;
END_VAR
VAR_OUTPUT
	
END_VAR
VAR
	
END_VAR

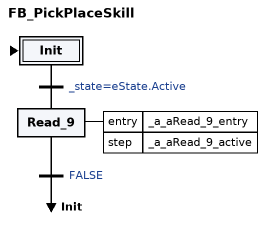
INITIAL_STEP Init:
END_STEP
TRANSITION FROM Init TO Read_9
    := _state=eState.Active;
END_TRANSITION
STEP Read_9:
    _a_aRead_9_entry(P1);  // entry action
    _a_aRead_9_active(N);  // step action
END_STEP
TRANSITION FROM Read_9 TO Init
    := FALSE;
END_TRANSITION

ACTION _a_aRead_9_active:

END_ACTION

ACTION _a_aRead_9_entry:
Rob^.MC_ReadDigitalInput(input:=8);
END_ACTION

END_FUNCTION_BLOCK

// ---- POUs/FB_ROB_MANIP.TcPOU
FUNCTION_BLOCK FB_ROB_MANIP EXTENDS FB_ROB IMPLEMENTS ITF_2_6AxisRobot



VAR_OUTPUT

END_VAR
VAR

	tcppos, tcpvel : stPose3D;
	jointpos, jointvel: stJoint6;
	currFrame: stFrame;
	currTool: FB_Tool;

END_VAR

//State Machine

{warning 'Add method implementation '}
METHOD M_Home : BOOL
END_METHOD

{warning 'Add method implementation '}
METHOD M_SwitchTool : UINT
VAR_INPUT
	tool	: FB_Tool;
END_VAR
END_METHOD

{warning 'Add method implementation '}
METHOD MC_MoveAxesAbsolute : BOOL
VAR_INPUT
	target	: stTarget3D;
END_VAR
IF _state=eState.Active THEN
// 	P_TargetReached:=FALSE;
END_IF
END_METHOD

{warning 'Add method implementation '}
METHOD MC_MoveAxesRelative : BOOL
VAR_INPUT
	axes	: ARRAY [1..6] OF FB_Axis;
	offsets	: ARRAY [1..6] OF REAL;
END_VAR
END_METHOD

{warning 'Add method implementation '}
METHOD MC_MoveLinearAbsolute : BOOL
VAR_INPUT
	target	: stTarget3D;
END_VAR
END_METHOD

{warning 'Add method implementation '}
METHOD MC_ReadActualVelocity : stPose
END_METHOD

{warning 'Add method implementation '}
METHOD MC_ReadAnalogInput : LREAL
VAR_INPUT
	input	: INT;
END_VAR
END_METHOD

{warning 'Add method implementation '}
METHOD MC_ReadDigitalInput : BOOL
VAR_INPUT
	input	: INT;
END_VAR
END_METHOD

{warning 'Add method implementation '}
METHOD MC_SetDigitalOutput : BOOL
VAR_INPUT
	output	: INT;
	value	: BOOL;
END_VAR
END_METHOD

{warning 'Add method implementation '}
METHOD MC_SetOperationMode : BOOL
VAR_INPUT
	mode	: eMode;
END_VAR
_mode:=mode;
END_METHOD

METHOD onActivate : BOOL
// ---- Init ----
transitionresult:=eResult.None;



// ---- Change ----

// _mode:= eMode.Automatic;




// ---- Check ----
transitionresult := eResult.SUCCESS;


// ---- Change State ----
IF transitionresult= eResult.SUCCESS THEN
	P_State:=eState.Active;
ELSIF transitionresult= eResult.FAILURE THEN
	P_State:=eState.Inactive;
ELSIF transitionresult= eResult.ERROR THEN
	P_State:=eState.ErrorProcessing;
ELSE
	ADSLOGSTR(ADSLOG_MSGTYPE_WARN,'Transitionresult from onActivate is None','');
END_IF
END_METHOD

METHOD onCleanup : BOOL
// ---- Init ----
transitionresult:=eResult.None;



// ---- Change ----

_mode:= eMode.Manual;




// ---- Check ----
transitionresult := eResult.SUCCESS;


// ---- Change State ----
IF transitionresult= eResult.SUCCESS THEN
	P_State:=eState.Unconfigured;
ELSIF transitionresult= eResult.FAILURE THEN
	ADSLOGSTR(ADSLOG_MSGTYPE_WARN,'Transitionresult from onCleanup is FAILURE ','');
ELSIF transitionresult= eResult.ERROR THEN
	P_State:=eState.ErrorProcessing;
ELSE
	ADSLOGSTR(ADSLOG_MSGTYPE_WARN,'Transitionresult from onCleanup is NONE','');
END_IF
END_METHOD

METHOD onConfigure : BOOL
// ---- Init ----
transitionresult:=eResult.None;



// ---- Change ----

_mode:= eMode.Manual;




// ---- Check ----
transitionresult := eResult.SUCCESS;


// ---- Change State ----
IF transitionresult= eResult.SUCCESS THEN
	P_State:=eState.Inactive;
ELSIF transitionresult= eResult.FAILURE THEN
	P_State:=eState.Unconfigured;
ELSIF transitionresult= eResult.ERROR THEN
	P_State:=eState.ErrorProcessing;
ELSE
	ADSLOGSTR(ADSLOG_MSGTYPE_WARN,'Transitionresult from onConfigure is None','');
END_IF
END_METHOD

METHOD onDeactivate : BOOL
// ---- Init ----
transitionresult:=eResult.None;



// ---- Change ----

_mode:= eMode.Manual;




// ---- Check ----
transitionresult := eResult.SUCCESS;


// ---- Change State ----
IF transitionresult= eResult.SUCCESS THEN
	P_State:=eState.Inactive;
ELSIF transitionresult= eResult.FAILURE THEN
	ADSLOGSTR(ADSLOG_MSGTYPE_WARN,'Transitionresult from onDeactivate is FAILURE','');
ELSIF transitionresult= eResult.ERROR THEN
	P_State:=eState.ErrorProcessing;
ELSE
	ADSLOGSTR(ADSLOG_MSGTYPE_WARN,'Transitionresult from onDeactivate is None','');
END_IF
END_METHOD

METHOD onError : BOOL
// ---- Init ----
transitionresult:=eResult.None;



// ---- Change ----

_mode:= eMode.Manual;




// ---- Check ----
transitionresult := eResult.SUCCESS;


// ---- Change State ----
IF transitionresult= eResult.SUCCESS THEN
	P_State:=eState.Unconfigured;
ELSIF transitionresult= eResult.FAILURE THEN
	P_State:=eState.Finalized;
ELSIF transitionresult= eResult.ERROR THEN
	ADSLOGSTR(ADSLOG_MSGTYPE_WARN,'Transitionresult from onError is Error','');
ELSE
	ADSLOGSTR(ADSLOG_MSGTYPE_WARN,'Transitionresult from onError is None','');
END_IF
END_METHOD

METHOD onShutdown : BOOL
// ---- Init ----
transitionresult:=eResult.None;



// ---- Change ----

_mode:= eMode.Manual;




// ---- Check ----
transitionresult := eResult.SUCCESS;


// ---- Change State ----
IF transitionresult= eResult.SUCCESS THEN
	P_State:=eState.Finalized;
ELSIF transitionresult= eResult.FAILURE THEN
	ADSLOGSTR(ADSLOG_MSGTYPE_WARN,'Transitionresult from onShutdown is FAILURE','');
ELSIF transitionresult= eResult.ERROR THEN
	P_State:=eState.ErrorProcessing;
ELSE
	ADSLOGSTR(ADSLOG_MSGTYPE_WARN,'Transitionresult from onShutdown is None','');
END_IF
END_METHOD

{warning 'Add property implementation'}
PROPERTY P_ActualAxisPos : stJoint6
GET
P_ActualAxisPos:= jointpos;
END_GET
END_PROPERTY

{warning 'Add property implementation'}
PROPERTY P_ActualJointVelocity : stJoint6
GET
P_ActualJointVelocity:= jointvel;
END_GET
END_PROPERTY

{warning 'Add property implementation'}
PROPERTY P_ActualTCPPos : stPose3D
GET
P_ActualTCPPos:=tcppos;
END_GET
END_PROPERTY

{warning 'Add property implementation'}
PROPERTY P_ActualTCPVelocity : stPose3D
GET
P_ActualTCPVelocity:=tcpvel;
END_GET
END_PROPERTY

{warning 'Add property implementation'}
PROPERTY P_currentFrame : stFrame
GET
P_currentFrame := currFrame;
END_GET
SET
currFrame := P_currentFrame;
END_SET
END_PROPERTY

{warning 'Add property implementation'}
PROPERTY P_currentFrameID : UINT
GET
P_currentFrameID:= currFrame.frameId;
END_GET
END_PROPERTY

{warning 'Add property implementation'}
PROPERTY P_currentTool : FB_Tool
GET
P_currentTool:= currTool;
END_GET
SET
currTool:= P_currentTool;
END_SET
END_PROPERTY

{warning 'Add property implementation'}
PROPERTY P_IsInHomePosition : BOOL
GET
END_GET
END_PROPERTY

PROPERTY P_TargetReached : BOOL
GET
END_GET
END_PROPERTY

END_FUNCTION_BLOCK

// ---- POUs/FB_Tool.TcPOU
FUNCTION_BLOCK FB_Tool EXTENDS FB_Base
VAR_INPUT
END_VAR
VAR_OUTPUT
END_VAR
VAR
END_VAR

METHOD onActivate : BOOL
// ---- Init ----
transitionresult:=eResult.None;



// ---- Change ----

// _mode:= eMode.Automatic;




// ---- Check ----
transitionresult := eResult.SUCCESS;


// ---- Change State ----
IF transitionresult= eResult.SUCCESS THEN
	P_State:=eState.Active;
ELSIF transitionresult= eResult.FAILURE THEN
	P_State:=eState.Inactive;
ELSIF transitionresult= eResult.ERROR THEN
	P_State:=eState.ErrorProcessing;
ELSE
	ADSLOGSTR(ADSLOG_MSGTYPE_WARN,'Transitionresult from onActivate is None','');
END_IF
END_METHOD

METHOD onCleanup : BOOL
// ---- Init ----
transitionresult:=eResult.None;



// ---- Change ----

// _mode:= eMode.Manual;




// ---- Check ----
transitionresult := eResult.SUCCESS;


// ---- Change State ----
IF transitionresult= eResult.SUCCESS THEN
	P_State:=eState.Unconfigured;
ELSIF transitionresult= eResult.FAILURE THEN
	ADSLOGSTR(ADSLOG_MSGTYPE_WARN,'Transitionresult from onCleanup is FAILURE ','');
ELSIF transitionresult= eResult.ERROR THEN
	P_State:=eState.ErrorProcessing;
ELSE
	ADSLOGSTR(ADSLOG_MSGTYPE_WARN,'Transitionresult from onCleanup is NONE','');
END_IF
END_METHOD

METHOD onConfigure : BOOL
// ---- Init ----
transitionresult:=eResult.None;



// ---- Change ----

// _mode:= eMode.Manual;




// ---- Check ----
transitionresult := eResult.SUCCESS;


// ---- Change State ----
IF transitionresult= eResult.SUCCESS THEN
	P_State:=eState.Inactive;
ELSIF transitionresult= eResult.FAILURE THEN
	P_State:=eState.Unconfigured;
ELSIF transitionresult= eResult.ERROR THEN
	P_State:=eState.ErrorProcessing;
ELSE
	ADSLOGSTR(ADSLOG_MSGTYPE_WARN,'Transitionresult from onConfigure is None','');
END_IF
END_METHOD

METHOD onDeactivate : BOOL
// ---- Init ----
transitionresult:=eResult.None;



// ---- Change ----

// _mode:= eMode.Manual;




// ---- Check ----
transitionresult := eResult.SUCCESS;


// ---- Change State ----
IF transitionresult= eResult.SUCCESS THEN
	P_State:=eState.Inactive;
ELSIF transitionresult= eResult.FAILURE THEN
	ADSLOGSTR(ADSLOG_MSGTYPE_WARN,'Transitionresult from onDeactivate is FAILURE','');
ELSIF transitionresult= eResult.ERROR THEN
	P_State:=eState.ErrorProcessing;
ELSE
	ADSLOGSTR(ADSLOG_MSGTYPE_WARN,'Transitionresult from onDeactivate is None','');
END_IF
END_METHOD

METHOD onError : BOOL
// ---- Init ----
transitionresult:=eResult.None;



// ---- Change ----

// _mode:= eMode.Manual;




// ---- Check ----
transitionresult := eResult.SUCCESS;


// ---- Change State ----
IF transitionresult= eResult.SUCCESS THEN
	P_State:=eState.Unconfigured;
ELSIF transitionresult= eResult.FAILURE THEN
	P_State:=eState.Finalized;
ELSIF transitionresult= eResult.ERROR THEN
	ADSLOGSTR(ADSLOG_MSGTYPE_WARN,'Transitionresult from onError is Error','');
ELSE
	ADSLOGSTR(ADSLOG_MSGTYPE_WARN,'Transitionresult from onError is None','');
END_IF
END_METHOD

METHOD onShutdown : BOOL
// ---- Init ----
transitionresult:=eResult.None;



// ---- Change ----

// _mode:= eMode.Manual;




// ---- Check ----
transitionresult := eResult.SUCCESS;


// ---- Change State ----
IF transitionresult= eResult.SUCCESS THEN
	P_State:=eState.Finalized;
ELSIF transitionresult= eResult.FAILURE THEN
	ADSLOGSTR(ADSLOG_MSGTYPE_WARN,'Transitionresult from onShutdown is FAILURE','');
ELSIF transitionresult= eResult.ERROR THEN
	P_State:=eState.ErrorProcessing;
ELSE
	ADSLOGSTR(ADSLOG_MSGTYPE_WARN,'Transitionresult from onShutdown is None','');
END_IF
END_METHOD

END_FUNCTION_BLOCK

// ---- POUs/Archiv/FB_Axis.TcPOU
FUNCTION_BLOCK FB_Axis EXTENDS FB_Base IMPLEMENTS ITF_0_BaseComponent
VAR_INPUT
END_VAR
VAR_OUTPUT
END_VAR
VAR
END_VAR

METHOD M_activate : BOOL
VAR_INPUT
END_VAR
END_METHOD

METHOD M_cleanup : BOOL
VAR_INPUT
END_VAR
END_METHOD

METHOD M_configure : BOOL
VAR_INPUT
END_VAR
END_METHOD

METHOD M_deactivate : BOOL
VAR_INPUT
END_VAR
END_METHOD

METHOD M_destroy : BOOL
VAR_INPUT
END_VAR
END_METHOD

METHOD M_shutdown : BOOL
VAR_INPUT
END_VAR
END_METHOD

METHOD onActivate : BOOL
VAR_INPUT
END_VAR
END_METHOD

METHOD onCleanup : BOOL
VAR_INPUT
END_VAR
END_METHOD

METHOD onConfigure : BOOL
VAR_INPUT
END_VAR
END_METHOD

METHOD onDeactivate : BOOL
VAR_INPUT
END_VAR
END_METHOD

METHOD onError : BOOL
VAR_INPUT
END_VAR
END_METHOD

METHOD onShutdown : BOOL
VAR_INPUT
END_VAR
END_METHOD

PROPERTY P_ID : UINT
GET
END_GET
SET
END_SET
END_PROPERTY

PROPERTY P_Name : String
GET
END_GET
END_PROPERTY

PROPERTY P_Path : String
GET
END_GET
END_PROPERTY

PROPERTY P_State : eState
GET
END_GET
SET
END_SET
END_PROPERTY

END_FUNCTION_BLOCK

// ---- POUs/FB_Helper.TcPOU
{attribute 'enable_dynamic_creation'}
FUNCTION_BLOCK FB_Helper
VAR
END_VAR

// Helper implementation

METHOD PUBLIC ImportConfigFromDB : BOOL
VAR_INPUT
	sFilePath : STRING(255);
END_VAR
// TODO: Implement file import
END_METHOD

METHOD PUBLIC LoadFrameConfigFromDB : BOOL
VAR_INPUT
	sFilePath : STRING(255);
END_VAR
// TODO: Implement frame config load
END_METHOD

METHOD PUBLIC LoadTargetConfigFromDB : BOOL
VAR_INPUT
	sFilePath : STRING(255);
END_VAR
// TODO: Implement target config load
END_METHOD

METHOD PUBLIC LoadToolConfigFromDB : BOOL
VAR_INPUT
	sFilePath : STRING(255);
END_VAR
// TODO: Implement tool config load
END_METHOD

METHOD PUBLIC SaveConfigToDB : BOOL
VAR_INPUT
	sFilePath : STRING(255);
END_VAR
// TODO: Implement file save
END_METHOD

METHOD PUBLIC SaveFrameConfigToDB : BOOL
VAR_INPUT
	sFilePath : STRING(255);
END_VAR
// TODO: Implement frame config save
END_METHOD

METHOD PUBLIC SaveTargetConfigToDB : BOOL
VAR_INPUT
	sFilePath : STRING(255);
END_VAR
// TODO: Implement target config save
END_METHOD

METHOD PUBLIC SaveToolConfigToDB : BOOL
VAR_INPUT
	sFilePath : STRING(255);
END_VAR
// TODO: Implement tool config save
END_METHOD

END_FUNCTION_BLOCK

// ---- POUs/FB_ROB_AMR.TcPOU
FUNCTION_BLOCK FB_ROB_AMR EXTENDS FB_ROB IMPLEMENTS  ITF_BA_AMR, ITF_2_AMR
VAR_INPUT
END_VAR
VAR_OUTPUT
END_VAR
VAR
		tcppos, tcpvel : stPose2D;
	jointpos, jointvel: stJoint2;
END_VAR

{warning 'Add method implementation '}
METHOD M_Dock : BOOL
END_METHOD

{error 'Add method implementation or delete method to use base implementation'}
METHOD MC_ChangeSpeedOverride : INT
VAR_INPUT
	factor	: REAL;
END_VAR
END_METHOD

{error 'Add method implementation or delete method to use base implementation'}
METHOD MC_MoveAxesAbsolute : BOOL
VAR_INPUT
	target	: stTarget3D;
END_VAR
END_METHOD

{error 'Add method implementation or delete method to use base implementation'}
METHOD MC_MoveAxesRelative : BOOL
VAR_INPUT
	axes	: ARRAY [1..6] OF FB_Axis;
	offsets	: ARRAY [1..6] OF REAL;
END_VAR
END_METHOD

{error 'Add method implementation or delete method to use base implementation'}
METHOD MC_MoveLinearAbsolute : BOOL
VAR_INPUT
	target	: stTarget3D;
END_VAR
END_METHOD

{error 'Add method implementation or delete method to use base implementation'}
METHOD MC_ReadAnalogInput : LREAL
VAR_INPUT
	input	: INT;
END_VAR
END_METHOD

{error 'Add method implementation or delete method to use base implementation'}
METHOD MC_ReadDigitalInput : BOOL
VAR_INPUT
	input	: INT;
END_VAR
END_METHOD

{error 'Add method implementation or delete method to use base implementation'}
METHOD MC_SetDigitalOutput : BOOL
VAR_INPUT
	output	: INT;
	value	: BOOL;
END_VAR
END_METHOD

{error 'Add method implementation or delete method to use base implementation'}
METHOD MC_SetOperationMode : BOOL
VAR_INPUT
	mode	: eMode;
END_VAR
END_METHOD

{warning 'Add property implementation'}
PROPERTY P_ActualAxisPos : stJoint2
GET
P_ActualAxisPos:= jointpos;
END_GET
END_PROPERTY

{warning 'Add property implementation'}
PROPERTY P_ActualJointVelocity : stJoint2
GET
P_ActualJointVelocity:= jointvel;
END_GET
END_PROPERTY

{warning 'Add property implementation'}
PROPERTY P_ActualTCPPos : stPose2D
GET
P_ActualTCPPos:=tcppos;
END_GET
END_PROPERTY

{warning 'Add property implementation'}
PROPERTY P_ActualTCPVelocity : stPose2D
GET
P_ActualTCPVelocity:=tcpvel;
END_GET
END_PROPERTY

{warning 'Add property implementation'}
PROPERTY P_IsDocked : BOOL
GET
END_GET
END_PROPERTY

{warning 'Add property implementation'}
PROPERTY P_RobotModel : STRING
GET
END_GET
END_PROPERTY

{error 'Add property implementation or delete property to use base implementation'}
PROPERTY P_TargetReached : BOOL
GET
END_GET
END_PROPERTY

END_FUNCTION_BLOCK

// ---- POUs/FB_UR5.TcPOU
FUNCTION_BLOCK FB_UR5 EXTENDS FB_ROB_MANIP IMPLEMENTS ITF_BA_6Axis, ITF_CommunicationModul
VAR_INPUT
END_VAR
VAR_OUTPUT
END_VAR
VAR
	PiNPl: FB_PickPlaceSkill;
END_VAR

StateMachine();


//Reference to Skills
PiNPl(Rob:=ADR(THIS^));

//ComConfig
ComConfig.sIPAdress:='127.0.0.1';
ComConfig.Port:= 5432;

METHOD M_Connect : BOOL
VAR_INPUT
END_VAR
END_METHOD

METHOD M_Disconnect : BOOL
VAR_INPUT
END_VAR
END_METHOD

METHOD M_ResetConnection : BOOL
VAR_INPUT
END_VAR
END_METHOD

{warning 'Add method implementation '}
METHOD MC_MoveAxesAbsolute : BOOL
VAR_INPUT
	target	: stTarget3D;
END_VAR
IF _state=eState.Active THEN
// 	P_TargetReached:=FALSE;
END_IF
END_METHOD

{warning 'Add method implementation '}
METHOD MC_MoveAxesRelative : BOOL
VAR_INPUT
	axes	: ARRAY [1..6] OF FB_Axis;
	offsets	: ARRAY [1..6] OF REAL;
END_VAR
END_METHOD

{warning 'Add method implementation '}
METHOD MC_MoveLinearAbsolute : BOOL
VAR_INPUT
	target	: stTarget3D;
END_VAR
END_METHOD

{warning 'Add method implementation '}
METHOD MC_ReadActualVelocity : stPose
END_METHOD

{warning 'Add method implementation '}
METHOD MC_ReadAnalogInput : LREAL
VAR_INPUT
	input	: INT;
END_VAR
END_METHOD

{warning 'Add method implementation '}
METHOD MC_ReadDigitalInput : BOOL
VAR_INPUT
	input	: INT;
END_VAR
END_METHOD

{warning 'Add method implementation '}
METHOD MC_SetDigitalOutput : BOOL
VAR_INPUT
	output	: INT;
	value	: BOOL;
END_VAR
END_METHOD

{warning 'Add method implementation '}
METHOD MC_SetOperationMode : BOOL
VAR_INPUT
	mode	: eMode;
END_VAR
_mode:=mode;
END_METHOD

PROPERTY P_bConnected : BOOL
GET
END_GET
END_PROPERTY

END_FUNCTION_BLOCK

// ---- POUs/MAIN_1.TcPOU
PROGRAM MAIN
VAR
	TestBot: FB_ROB;
	H: FB_HELPER;
	UR5: FB_UR5;
	PnP : FB_PickPlaceSkill;
END_VAR


VAR

    fbDB : FB_PostgreSQLClient;


    sRobotName : STRING;


END_VAR

fbDB();

// PnP(Rob:=ADR(UR5));
UR5();

UR5.CallSkill(pSkill:=ADR(UR5.PiNPl));

END_PROGRAM

// ---- POUs/Robots/FB_OmronLD90.TcPOU
FUNCTION_BLOCK FB_OmronLD90 EXTENDS FB_ROB_AMR IMPLEMENTS 
VAR_INPUT
END_VAR
VAR_OUTPUT
END_VAR
VAR
	//Reference to Skills

END_VAR

StateMachine(); // Method in FB_Base
ComMachine();	//Method in FB_ROB
DBClient();	//Datenbank Client in FB_ROB


PiNPl(Rob:=ADR(THIS^));

METHOD ComMachine : BOOL
VAR_INPUT
END_VAR
CASE eConnectionState OF


    // =========================================================
    // DISCONNECTED
    // =========================================================

    eCommunicationState.DISCONNECTED:

       _connected := FALSE;


        // Make sure socket handle is cleared
//         hSocket


        // -----------------------------------------------------
        // Connect requested
        // -----------------------------------------------------

        IF xConnectRequest THEN

            xConnectRequest := FALSE;

            // Clear previous errors
            Error := FALSE;
            ErrorId := 0;
            SocketErrorId := 0;

            // Start FB_SocketConnect
            xSocketConnectExecute := TRUE;

            eConnectionState :=
                eCommunicationState.CONNECTING;

        END_IF;


    // =========================================================
    // CONNECTING
    // =========================================================

    eCommunicationState.CONNECTING:

        _connected := FALSE;
        


        // -----------------------------------------------------
        // Execute FB_SocketConnect
        // -----------------------------------------------------

        fbSocketConnect(
            sSrvNetId := '',
            sRemoteHost := ComConfig.sIpAddress,
            nRemotePort := ComConfig.nPort,
            bExecute := xSocketConnectExecute,
            tTimeout := ComConfig.tTimeout
        );


        // Execute must only be TRUE for one cycle
        xSocketConnectExecute := FALSE;


        // -----------------------------------------------------
        // Connection successful
        // -----------------------------------------------------

        IF NOT fbSocketConnect.bBusy
            AND NOT fbSocketConnect.bError
//             AND (fbSocketConnect.hSocket <> 0)
        THEN

            hSocket :=
                fbSocketConnect.hSocket;

            _connected := TRUE;
    

            Error := FALSE;
            ErrorId := 0;
            SocketErrorId := 0;

            eConnectionState :=
                eCommunicationState.CONNECTED;

        END_IF;


        // -----------------------------------------------------
        // Connection failed
        // -----------------------------------------------------

        IF NOT fbSocketConnect.bBusy
            AND fbSocketConnect.bError
        THEN

            _connected := FALSE;

            Error := TRUE;

            SocketErrorId :=
                fbSocketConnect.nErrId;

            ErrorId :=
                fbSocketConnect.nErrId;

//             hSocket := 0;

            eConnectionState :=
                eCommunicationState.ERROR;

        END_IF;


    // =========================================================
    // CONNECTED
    // =========================================================

    eCommunicationState.CONNECTED:

        _connected := TRUE;



        // -----------------------------------------------------
        // Disconnect requested
        // -----------------------------------------------------

        IF xDisconnectRequest THEN

            xDisconnectRequest := FALSE;


            // Start socket close
            xSocketCloseExecute := TRUE;

            eConnectionState :=
                eCommunicationState.DISCONNECTING;

        END_IF;


    // =========================================================
    // DISCONNECTING
    // =========================================================

    eCommunicationState.DISCONNECTING:

        _connected := FALSE;


        // -----------------------------------------------------
        // Execute FB_SocketClose
        // -----------------------------------------------------

        fbSocketClose(
            sSrvNetId := '',
            hSocket := hSocket,
            bExecute := xSocketCloseExecute,
            tTimeout := ComConfig.tTimeout
        );


        // Execute only for one cycle
        xSocketCloseExecute := FALSE;


        // -----------------------------------------------------
        // Socket closed successfully
        // -----------------------------------------------------

        IF NOT fbSocketClose.bBusy
            AND NOT fbSocketClose.bError
        THEN

            _connected := FALSE;


//             hSocket := 0;

            eConnectionState :=
                eCommunicationState.DISCONNECTED;

        END_IF;


        // -----------------------------------------------------
        // Socket close failed
        // -----------------------------------------------------

        IF NOT fbSocketClose.bBusy
            AND fbSocketClose.bError
        THEN

            _connected := FALSE;


            Error := TRUE;

            SocketErrorId :=
                fbSocketClose.nErrId;

            ErrorId :=
                fbSocketClose.nErrId;

            // The socket should no longer be used
//             hSocket := 0;

            eConnectionState :=
                eCommunicationState.ERROR;

        END_IF;


    // =========================================================
    // ERROR
    // =========================================================

    eCommunicationState.ERROR:

        _connected := FALSE;
        // -----------------------------------------------------
        // Do not attempt to use the socket after an error
        // -----------------------------------------------------

//         hSocket := 0;


        // -----------------------------------------------------
        // A new connection request can recover from the error
        // -----------------------------------------------------

        IF xConnectRequest THEN

            xConnectRequest := FALSE;

            Error := FALSE;
            ErrorId := 0;
            SocketErrorId := 0;

            xSocketConnectExecute := TRUE;

            eConnectionState :=
                eCommunicationState.CONNECTING;

        END_IF;


END_CASE;
END_METHOD

{warning 'Add method implementation '}
METHOD Connect : BOOL

Connect := FALSE;

// Already connected
IF eConnectionState = eCommunicationState.CONNECTED THEN
    Connect := TRUE;
    RETURN;
END_IF;

// Already trying to connect
IF eConnectionState = eCommunicationState.CONNECTING THEN
    Connect := TRUE;
    RETURN;
END_IF;

// Don't accept a new connection while disconnecting
IF eConnectionState = eCommunicationState.DISCONNECTING THEN
    RETURN;
END_IF;

// Validate address
IF LEN(ComConfig.sIpAddress) = 0 THEN
    Error := TRUE;
//     ErrorId := 16#1001;
    RETURN;
END_IF;

// Validate port
IF ComConfig.nPort = 0 THEN
    Error := TRUE;
//     ErrorId := 16#1002;
    RETURN;
END_IF;

// Clear previous error
Error := FALSE;
ErrorId := 0;

// Request connection
xConnectRequest := TRUE;

Connect := TRUE;
END_METHOD

{warning 'Add property implementation'}
PROPERTY Connected : BOOL
GET
Connected:=_connected;
END_GET
END_PROPERTY

{warning 'Add method implementation '}
METHOD Disconnect : BOOL
END_METHOD

METHOD Dock : BOOL
END_METHOD

{warning 'Add method implementation '}
METHOD FINAL GoToGoal : BOOL
VAR_INPUT
	Goal: STRING;
END_VAR
END_METHOD

{warning 'Add method implementation '}
METHOD GoToPoint : BOOL

VAR_INPUT
	rX, rY, rTheta: REAL;
END_VAR
END_METHOD

METHOD MC_ChangeSpeedOverride : INT
VAR_INPUT
	factor	: REAL;
END_VAR
END_METHOD

METHOD MC_MoveAxesAbsolute : BOOL
VAR_INPUT
	target	: stTarget3D;
END_VAR
END_METHOD

METHOD MC_MoveAxesRelative : BOOL
VAR_INPUT
	axes	: ARRAY [1..6] OF FB_Axis;
	offsets	: ARRAY [1..6] OF REAL;
END_VAR
END_METHOD

METHOD MC_MoveLinearAbsolute : BOOL
VAR_INPUT
	target	: stTarget3D;
END_VAR
END_METHOD

METHOD MC_ReadAnalogInput : LREAL
VAR_INPUT
	input	: INT;
END_VAR
END_METHOD

METHOD MC_ReadDigitalInput : BOOL
VAR_INPUT
	input	: INT;
END_VAR
END_METHOD

METHOD MC_SetDigitalOutput : BOOL
VAR_INPUT
	output	: INT;
	value	: BOOL;
END_VAR
END_METHOD

METHOD MC_SetOperationMode : BOOL
VAR_INPUT
	mode	: eMode;
END_VAR
END_METHOD

METHOD onActivate : BOOL
// ---- Init ----
transitionresult:=eResult.None;



// ---- Change ----

// _mode:= eMode.Automatic;




// ---- Check ----
transitionresult := eResult.SUCCESS;

IF Error THEN
	transitionresult:= eResult.ERROR;
END_IF


// ---- Change State ----
IF transitionresult= eResult.SUCCESS THEN
	State:=eState.Active;
ELSIF transitionresult= eResult.FAILURE THEN
	State:=eState.Inactive;
ELSIF transitionresult= eResult.ERROR THEN
	State:=eState.ErrorProcessing;
ELSE
	ADSLOGSTR(ADSLOG_MSGTYPE_WARN,'Transitionresult from onActivate is None','');
END_IF
END_METHOD

METHOD onCleanup : BOOL
// ---- Init ----
transitionresult:=eResult.None;



// ---- Change ----

IF Connected THEN
	Disconnect();
END_IF





// ---- Check ----
transitionresult := eResult.SUCCESS;


// ---- Change State ----
IF transitionresult= eResult.SUCCESS THEN
	State:=eState.Unconfigured;
ELSIF transitionresult= eResult.FAILURE THEN
	ADSLOGSTR(ADSLOG_MSGTYPE_WARN,'Transitionresult from onCleanup is FAILURE ','');
ELSIF transitionresult= eResult.ERROR THEN
	State:=eState.ErrorProcessing;
ELSE
	ADSLOGSTR(ADSLOG_MSGTYPE_WARN,'Transitionresult from onCleanup is NONE','');
END_IF
END_METHOD

METHOD onConfigure : BOOL
// ---- Init ----
transitionresult:=eResult.None;



// ---- Change ----

Connect();




// ---- Check ----
IF Connected THEN
	transitionresult := eResult.SUCCESS;
ELSE
	transitionresult := eResult.FAILURE;
END_IF

IF Error THEN
	transitionresult:= eResult.ERROR;
END_IF



// ---- Change State ----
IF transitionresult= eResult.SUCCESS THEN
	State:=eState.Inactive;
ELSIF transitionresult= eResult.FAILURE THEN
	State:=eState.Unconfigured;
ELSIF transitionresult= eResult.ERROR THEN
	State:=eState.ErrorProcessing;
ELSE
	ADSLOGSTR(ADSLOG_MSGTYPE_WARN,'Transitionresult from onConfigure is None','');
END_IF
END_METHOD

METHOD onDeactivate : BOOL
// ---- Init ----
transitionresult:=eResult.None;



// ---- Change ----

// _mode:= eMode.Manual;




// ---- Check ----
transitionresult := eResult.SUCCESS;

IF Error THEN
	transitionresult:= eResult.ERROR;
END_IF

// ---- Change State ----
IF transitionresult= eResult.SUCCESS THEN
	State:=eState.Inactive;
ELSIF transitionresult= eResult.FAILURE THEN
	ADSLOGSTR(ADSLOG_MSGTYPE_WARN,'Transitionresult from onDeactivate is FAILURE','');
ELSIF transitionresult= eResult.ERROR THEN
	State:=eState.ErrorProcessing;
ELSE
	ADSLOGSTR(ADSLOG_MSGTYPE_WARN,'Transitionresult from onDeactivate is None','');
END_IF
END_METHOD

METHOD onError : BOOL
// ---- Init ----
transitionresult:=eResult.None;



// ---- Change ----

// _mode:= eMode.Manual;




// ---- Check ----
transitionresult := eResult.SUCCESS;


// ---- Change State ----
IF transitionresult= eResult.SUCCESS THEN
	State:=eState.Unconfigured;
ELSIF transitionresult= eResult.FAILURE THEN
	State:=eState.Finalized;
ELSIF transitionresult= eResult.ERROR THEN
	ADSLOGSTR(ADSLOG_MSGTYPE_WARN,'Transitionresult from onError is Error','');
ELSE
	ADSLOGSTR(ADSLOG_MSGTYPE_WARN,'Transitionresult from onError is None','');
END_IF
END_METHOD

METHOD onShutdown : BOOL
// ---- Init ----
transitionresult:=eResult.None;



// ---- Change ----

// _mode:= eMode.Manual;

IF Connected THEN
	Disconnect();
END_IF


// ---- Check ----
transitionresult := eResult.SUCCESS;

IF Error THEN
	transitionresult:= eResult.ERROR;
END_IF

// ---- Change State ----
IF transitionresult= eResult.SUCCESS THEN
	State:=eState.Finalized;
ELSIF transitionresult= eResult.FAILURE THEN
	ADSLOGSTR(ADSLOG_MSGTYPE_WARN,'Transitionresult from onShutdown is FAILURE','');
ELSIF transitionresult= eResult.ERROR THEN
	State:=eState.ErrorProcessing;
ELSE
	ADSLOGSTR(ADSLOG_MSGTYPE_WARN,'Transitionresult from onShutdown is None','');
END_IF
END_METHOD

{warning 'Add method implementation '}
METHOD ResetConnection : BOOL
END_METHOD

{warning 'Add method implementation '}
METHOD Undock : BOOL
END_METHOD

END_FUNCTION_BLOCK

// ---- POUs/Robots/FB_ROB_1.TcPOU
FUNCTION_BLOCK FB_ROB EXTENDS FB_Base IMPLEMENTS ITF_1_Robot, ITF_CommunicationModul

VAR_INPUT
	Skills: ARRAY[1..3] OF FB_Skill;
	SH: FB_SkillHandler;
END_VAR

VAR_INPUT
	ComConfig: ST_CommunicationConfig;

END_VAR


VAR_OUTPUT
	_inCollision: BOOL;
	 eConnectionState : eCommunicationState :=
        eCommunicationState.DISCONNECTED;
END_VAR
VAR
	    // ============================================================
    // Internal state
    // ============================================================

    _Connected : BOOL;
    _Busy : BOOL;


    _Command : STRING(1023);
    _CommandPending : BOOL;

    _ReconnectTimer : TON;
    _TimeoutTimer : TON;


    // Rising-edge detection
	
    _ExecuteConnect : BOOL;
    _ExecuteDisconnect : BOOL;
    _ExecuteCommand : BOOL;

    _LastCommand : STRING(1023);
	
	
	_enabled: BOOL;
	_mode: eMode;
	_locked: BOOL;
	
	velovr: BOOL;
	velfact: REAL;
	
	DBClient: FB_PostgreSQLClient;
	

END_VAR


VAR
    // =========================================================
    // Communication state
    // =========================================================

   

    xConnectRequest : BOOL := FALSE;
    xDisconnectRequest : BOOL := FALSE;

    // One-shot execute signals
    xSocketConnectExecute : BOOL := FALSE;
    xSocketCloseExecute : BOOL := FALSE;


    fbSocketConnect : FB_SocketConnect;
    fbSocketClose : FB_SocketClose;

    hSocket : T_HSOCKET;


    SocketErrorId : UDINT := 0;
END_VAR

//State Machine
ComMachine();
DBClient();

METHOD ComMachine : BOOL
VAR_INPUT
END_VAR
CASE eConnectionState OF


    // =========================================================
    // DISCONNECTED
    // =========================================================

    eCommunicationState.DISCONNECTED:

       _connected := FALSE;


        // Make sure socket handle is cleared
//         hSocket


        // -----------------------------------------------------
        // Connect requested
        // -----------------------------------------------------

        IF xConnectRequest THEN

            xConnectRequest := FALSE;

            // Clear previous errors
            Error := FALSE;
            ErrorId := 0;
            SocketErrorId := 0;

            // Start FB_SocketConnect
            xSocketConnectExecute := TRUE;

            eConnectionState :=
                eCommunicationState.CONNECTING;

        END_IF;


    // =========================================================
    // CONNECTING
    // =========================================================

    eCommunicationState.CONNECTING:

        _connected := FALSE;
        


        // -----------------------------------------------------
        // Execute FB_SocketConnect
        // -----------------------------------------------------

        fbSocketConnect(
            sSrvNetId := '',
            sRemoteHost := ComConfig.sIpAddress,
            nRemotePort := ComConfig.nPort,
            bExecute := xSocketConnectExecute,
            tTimeout := ComConfig.tTimeout
        );


        // Execute must only be TRUE for one cycle
        xSocketConnectExecute := FALSE;


        // -----------------------------------------------------
        // Connection successful
        // -----------------------------------------------------

        IF NOT fbSocketConnect.bBusy
            AND NOT fbSocketConnect.bError
//             AND (fbSocketConnect.hSocket <> 0)
        THEN

            hSocket :=
                fbSocketConnect.hSocket;

            _connected := TRUE;
    

            Error := FALSE;
            ErrorId := 0;
            SocketErrorId := 0;

            eConnectionState :=
                eCommunicationState.CONNECTED;

        END_IF;


        // -----------------------------------------------------
        // Connection failed
        // -----------------------------------------------------

        IF NOT fbSocketConnect.bBusy
            AND fbSocketConnect.bError
        THEN

            _connected := FALSE;

            Error := TRUE;

            SocketErrorId :=
                fbSocketConnect.nErrId;

            ErrorId :=
                fbSocketConnect.nErrId;

//             hSocket := 0;

            eConnectionState :=
                eCommunicationState.ERROR;

        END_IF;


    // =========================================================
    // CONNECTED
    // =========================================================

    eCommunicationState.CONNECTED:

        _connected := TRUE;



        // -----------------------------------------------------
        // Disconnect requested
        // -----------------------------------------------------

        IF xDisconnectRequest THEN

            xDisconnectRequest := FALSE;


            // Start socket close
            xSocketCloseExecute := TRUE;

            eConnectionState :=
                eCommunicationState.DISCONNECTING;

        END_IF;


    // =========================================================
    // DISCONNECTING
    // =========================================================

    eCommunicationState.DISCONNECTING:

        _connected := FALSE;


        // -----------------------------------------------------
        // Execute FB_SocketClose
        // -----------------------------------------------------

        fbSocketClose(
            sSrvNetId := '',
            hSocket := hSocket,
            bExecute := xSocketCloseExecute,
            tTimeout := ComConfig.tTimeout
        );


        // Execute only for one cycle
        xSocketCloseExecute := FALSE;


        // -----------------------------------------------------
        // Socket closed successfully
        // -----------------------------------------------------

        IF NOT fbSocketClose.bBusy
            AND NOT fbSocketClose.bError
        THEN

            _connected := FALSE;


//             hSocket := 0;

            eConnectionState :=
                eCommunicationState.DISCONNECTED;

        END_IF;


        // -----------------------------------------------------
        // Socket close failed
        // -----------------------------------------------------

        IF NOT fbSocketClose.bBusy
            AND fbSocketClose.bError
        THEN

            _connected := FALSE;


            Error := TRUE;

            SocketErrorId :=
                fbSocketClose.nErrId;

            ErrorId :=
                fbSocketClose.nErrId;

            // The socket should no longer be used
//             hSocket := 0;

            eConnectionState :=
                eCommunicationState.ERROR;

        END_IF;


    // =========================================================
    // ERROR
    // =========================================================

    eCommunicationState.ERROR:

        _connected := FALSE;
        // -----------------------------------------------------
        // Do not attempt to use the socket after an error
        // -----------------------------------------------------

//         hSocket := 0;


        // -----------------------------------------------------
        // A new connection request can recover from the error
        // -----------------------------------------------------

        IF xConnectRequest THEN

            xConnectRequest := FALSE;

            Error := FALSE;
            ErrorId := 0;
            SocketErrorId := 0;

            xSocketConnectExecute := TRUE;

            eConnectionState :=
                eCommunicationState.CONNECTING;

        END_IF;


END_CASE;
END_METHOD

{warning 'Add method implementation '}
METHOD Connect : BOOL

Connect := FALSE;

// Already connected
IF eConnectionState = eCommunicationState.CONNECTED THEN
    Connect := TRUE;
    RETURN;
END_IF;

// Already trying to connect
IF eConnectionState = eCommunicationState.CONNECTING THEN
    Connect := TRUE;
    RETURN;
END_IF;

// Don't accept a new connection while disconnecting
IF eConnectionState = eCommunicationState.DISCONNECTING THEN
    RETURN;
END_IF;

// Validate address
IF LEN(ComConfig.sIpAddress) = 0 THEN
    Error := TRUE;
//     ErrorId := 16#1001;
    RETURN;
END_IF;

// Validate port
IF ComConfig.nPort = 0 THEN
    Error := TRUE;
//     ErrorId := 16#1002;
    RETURN;
END_IF;

// Clear previous error
Error := FALSE;
ErrorId := 0;

// Request connection
xConnectRequest := TRUE;

Connect := TRUE;
END_METHOD

{warning 'Add property implementation'}
PROPERTY Connected : BOOL
GET
Connected:=_connected;
END_GET
END_PROPERTY

{warning 'Add method implementation '}
METHOD Disconnect : BOOL
END_METHOD

{warning 'Add method implementation '}
METHOD M_AUTO : BOOL
_mode:=eMode.Automatic;
END_METHOD

{warning 'Add method implementation '}
METHOD M_Disable : BOOL
_enabled:=FALSE;
super^.Deactivate();
END_METHOD

{warning 'Add method implementation '}
METHOD M_DisableVelocityOverride : BOOL
velovr:=False;
END_METHOD

{warning 'Add method implementation '}
METHOD M_Enable : BOOL
_enabled:=TRUE;
END_METHOD

{warning 'Add method implementation '}
METHOD M_EnableVelocityOverride : BOOL
velovr:=True;
END_METHOD

{warning 'Add method implementation '}
METHOD M_EStop : BOOL
END_METHOD

{warning 'Add method implementation '}
METHOD M_MAN : BOOL
_mode:=eMode.Manual;
END_METHOD

{warning 'Add method implementation '}
METHOD MC_ChangeSpeedOverride : INT
VAR_INPUT
	factor	: REAL;
END_VAR
velfact:=factor;
END_METHOD

METHOD onActivate : BOOL
// ---- Init ----
transitionresult:=eResult.None;



// ---- Change ----

// _mode:= eMode.Automatic;




// ---- Check ----
transitionresult := eResult.SUCCESS;


// ---- Change State ----
IF transitionresult= eResult.SUCCESS THEN
	State:=eState.Active;
ELSIF transitionresult= eResult.FAILURE THEN
	State:=eState.Inactive;
ELSIF transitionresult= eResult.ERROR THEN
	State:=eState.ErrorProcessing;
ELSE
	ADSLOGSTR(ADSLOG_MSGTYPE_WARN,'Transitionresult from onActivate is None','');
END_IF
END_METHOD

METHOD onCleanup : BOOL
// ---- Init ----
transitionresult:=eResult.None;



// ---- Change ----

_mode:= eMode.Manual;




// ---- Check ----
transitionresult := eResult.SUCCESS;


// ---- Change State ----
IF transitionresult= eResult.SUCCESS THEN
	State:=eState.Unconfigured;
ELSIF transitionresult= eResult.FAILURE THEN
	ADSLOGSTR(ADSLOG_MSGTYPE_WARN,'Transitionresult from onCleanup is FAILURE ','');
ELSIF transitionresult= eResult.ERROR THEN
	State:=eState.ErrorProcessing;
ELSE
	ADSLOGSTR(ADSLOG_MSGTYPE_WARN,'Transitionresult from onCleanup is NONE','');
END_IF
END_METHOD

METHOD onConfigure : BOOL
// ---- Init ----
transitionresult:=eResult.None;



// ---- Change ----

_mode:= eMode.Manual;




// ---- Check ----
transitionresult := eResult.SUCCESS;


// ---- Change State ----
IF transitionresult= eResult.SUCCESS THEN
	State:=eState.Inactive;
ELSIF transitionresult= eResult.FAILURE THEN
	State:=eState.Unconfigured;
ELSIF transitionresult= eResult.ERROR THEN
	State:=eState.ErrorProcessing;
ELSE
	ADSLOGSTR(ADSLOG_MSGTYPE_WARN,'Transitionresult from onConfigure is None','');
END_IF
END_METHOD

METHOD onDeactivate : BOOL
// ---- Init ----
transitionresult:=eResult.None;



// ---- Change ----

_mode:= eMode.Manual;




// ---- Check ----
transitionresult := eResult.SUCCESS;


// ---- Change State ----
IF transitionresult= eResult.SUCCESS THEN
	State:=eState.Inactive;
ELSIF transitionresult= eResult.FAILURE THEN
	ADSLOGSTR(ADSLOG_MSGTYPE_WARN,'Transitionresult from onDeactivate is FAILURE','');
ELSIF transitionresult= eResult.ERROR THEN
	State:=eState.ErrorProcessing;
ELSE
	ADSLOGSTR(ADSLOG_MSGTYPE_WARN,'Transitionresult from onDeactivate is None','');
END_IF
END_METHOD

METHOD onError : BOOL
// ---- Init ----
transitionresult:=eResult.None;



// ---- Change ----

_mode:= eMode.Manual;




// ---- Check ----
transitionresult := eResult.SUCCESS;


// ---- Change State ----
IF transitionresult= eResult.SUCCESS THEN
	State:=eState.Unconfigured;
ELSIF transitionresult= eResult.FAILURE THEN
	State:=eState.Finalized;
ELSIF transitionresult= eResult.ERROR THEN
	ADSLOGSTR(ADSLOG_MSGTYPE_WARN,'Transitionresult from onError is Error','');
ELSE
	ADSLOGSTR(ADSLOG_MSGTYPE_WARN,'Transitionresult from onError is None','');
END_IF
END_METHOD

METHOD onShutdown : BOOL
// ---- Init ----
transitionresult:=eResult.None;



// ---- Change ----

_mode:= eMode.Manual;




// ---- Check ----
transitionresult := eResult.SUCCESS;


// ---- Change State ----
IF transitionresult= eResult.SUCCESS THEN
	State:=eState.Finalized;
ELSIF transitionresult= eResult.FAILURE THEN
	ADSLOGSTR(ADSLOG_MSGTYPE_WARN,'Transitionresult from onShutdown is FAILURE','');
ELSIF transitionresult= eResult.ERROR THEN
	State:=eState.ErrorProcessing;
ELSE
	ADSLOGSTR(ADSLOG_MSGTYPE_WARN,'Transitionresult from onShutdown is None','');
END_IF
END_METHOD

{warning 'Add property implementation'}
PROPERTY P_isInCollision : BOOL
GET
P_isInCollision:=_inCollision;
END_GET
END_PROPERTY

{warning 'Add property implementation'}
PROPERTY P_JogSpeed : LREAL
GET
END_GET
SET
END_SET
END_PROPERTY

{warning 'Add property implementation'}
PROPERTY P_RobotIsMoving : BOOL
GET
END_GET
END_PROPERTY

{warning 'Add property implementation'}
PROPERTY P_RobotIsReady : BOOL
GET
END_GET
END_PROPERTY

{warning 'Add method implementation '}
METHOD ResetConnection : BOOL
END_METHOD

END_FUNCTION_BLOCK

// ---- POUs/Robots/FB_ROB_AMR_1.TcPOU
FUNCTION_BLOCK FB_ROB_AMR EXTENDS FB_ROB IMPLEMENTS ITF_2_AMR, ITF_BA_AMR
VAR_INPUT
END_VAR
VAR_OUTPUT
END_VAR
VAR
	tcppos, tcpvel : stPose2D;
	jointpos, jointvel: stJoint2;
END_VAR

{warning 'Add property implementation'}
PROPERTY ActualAxisPos : stJoint2
GET
ActualAxisPos:= jointpos;
END_GET
END_PROPERTY

{warning 'Add property implementation'}
PROPERTY ActualJointVelocity : stJoint2
GET
ActualJointVelocity:= jointvel;
END_GET
END_PROPERTY

{warning 'Add property implementation'}
PROPERTY ActualTCPPos : stPose2D
GET
ActualTCPPos:=tcppos;
END_GET
END_PROPERTY

{warning 'Add property implementation'}
PROPERTY ActualTCPVelocity : stPose2D
GET
ActualTCPVelocity:=tcpvel;
END_GET
END_PROPERTY

METHOD Dock : BOOL
END_METHOD

{warning 'Add method implementation '}
METHOD GoToGoal : BOOL
VAR_INPUT
	Goal: STRING;
END_VAR
END_METHOD

{warning 'Add method implementation '}
METHOD GoToPoint : BOOL

VAR_INPUT
	rX, rY, rTheta: REAL;
END_VAR
END_METHOD

{warning 'Add property implementation'}
PROPERTY IsDocked : BOOL
GET
END_GET
END_PROPERTY

METHOD MC_ChangeSpeedOverride : INT
VAR_INPUT
	factor	: REAL;
END_VAR
END_METHOD

METHOD MC_MoveAxesAbsolute : BOOL
VAR_INPUT
	target	: stTarget3D;
END_VAR
END_METHOD

METHOD MC_MoveAxesRelative : BOOL
VAR_INPUT
	axes	: ARRAY [1..6] OF FB_Axis;
	offsets	: ARRAY [1..6] OF REAL;
END_VAR
END_METHOD

METHOD MC_MoveLinearAbsolute : BOOL
VAR_INPUT
	target	: stTarget3D;
END_VAR
END_METHOD

METHOD MC_ReadAnalogInput : LREAL
VAR_INPUT
	input	: INT;
END_VAR
END_METHOD

METHOD MC_ReadDigitalInput : BOOL
VAR_INPUT
	input	: INT;
END_VAR
END_METHOD

METHOD MC_SetDigitalOutput : BOOL
VAR_INPUT
	output	: INT;
	value	: BOOL;
END_VAR
END_METHOD

METHOD MC_SetOperationMode : BOOL
VAR_INPUT
	mode	: eMode;
END_VAR
END_METHOD

PROPERTY TargetReached : BOOL
GET
END_GET
END_PROPERTY

{warning 'Add method implementation '}
METHOD Undock : BOOL
END_METHOD

END_FUNCTION_BLOCK

// ---- POUs/Robots/FB_ROB_MANIP_1.TcPOU
FUNCTION_BLOCK FB_ROB_MANIP EXTENDS FB_ROB IMPLEMENTS ITF_2_6AxisRobot



VAR_OUTPUT

END_VAR
VAR

	tcppos, tcpvel : stPose3D;
	jointpos, jointvel: stJoint6;
	currFrame: stFrame;
	currTool: FB_Tool;

END_VAR

//State Machine

{warning 'Add method implementation '}
METHOD M_Home : BOOL
END_METHOD

{warning 'Add method implementation '}
METHOD M_SwitchTool : UINT
VAR_INPUT
	tool	: FB_Tool;
END_VAR
END_METHOD

{warning 'Add method implementation '}
METHOD MC_MoveAxesAbsolute : BOOL
VAR_INPUT
	target	: stTarget3D;
END_VAR
IF _state=eState.Active THEN
// 	P_TargetReached:=FALSE;
END_IF
END_METHOD

{warning 'Add method implementation '}
METHOD MC_MoveAxesRelative : BOOL
VAR_INPUT
	axes	: ARRAY [1..6] OF FB_Axis;
	offsets	: ARRAY [1..6] OF REAL;
END_VAR
END_METHOD

{warning 'Add method implementation '}
METHOD MC_MoveLinearAbsolute : BOOL
VAR_INPUT
	target	: stTarget3D;
END_VAR
END_METHOD

{warning 'Add method implementation '}
METHOD MC_ReadActualVelocity : stPose
END_METHOD

{warning 'Add method implementation '}
METHOD MC_ReadAnalogInput : LREAL
VAR_INPUT
	input	: INT;
END_VAR
END_METHOD

{warning 'Add method implementation '}
METHOD MC_ReadDigitalInput : BOOL
VAR_INPUT
	input	: INT;
END_VAR
END_METHOD

{warning 'Add method implementation '}
METHOD MC_SetDigitalOutput : BOOL
VAR_INPUT
	output	: INT;
	value	: BOOL;
END_VAR
END_METHOD

{warning 'Add method implementation '}
METHOD MC_SetOperationMode : BOOL
VAR_INPUT
	mode	: eMode;
END_VAR
_mode:=mode;
END_METHOD

METHOD onActivate : BOOL
// ---- Init ----
transitionresult:=eResult.None;



// ---- Change ----

// _mode:= eMode.Automatic;




// ---- Check ----
transitionresult := eResult.SUCCESS;


// ---- Change State ----
IF transitionresult= eResult.SUCCESS THEN
	State:=eState.Active;
ELSIF transitionresult= eResult.FAILURE THEN
	State:=eState.Inactive;
ELSIF transitionresult= eResult.ERROR THEN
	State:=eState.ErrorProcessing;
ELSE
	ADSLOGSTR(ADSLOG_MSGTYPE_WARN,'Transitionresult from onActivate is None','');
END_IF
END_METHOD

METHOD onCleanup : BOOL
// ---- Init ----
transitionresult:=eResult.None;



// ---- Change ----

_mode:= eMode.Manual;




// ---- Check ----
transitionresult := eResult.SUCCESS;


// ---- Change State ----
IF transitionresult= eResult.SUCCESS THEN
	State:=eState.Unconfigured;
ELSIF transitionresult= eResult.FAILURE THEN
	ADSLOGSTR(ADSLOG_MSGTYPE_WARN,'Transitionresult from onCleanup is FAILURE ','');
ELSIF transitionresult= eResult.ERROR THEN
	State:=eState.ErrorProcessing;
ELSE
	ADSLOGSTR(ADSLOG_MSGTYPE_WARN,'Transitionresult from onCleanup is NONE','');
END_IF
END_METHOD

METHOD onConfigure : BOOL
// ---- Init ----
transitionresult:=eResult.None;



// ---- Change ----

_mode:= eMode.Manual;




// ---- Check ----
transitionresult := eResult.SUCCESS;


// ---- Change State ----
IF transitionresult= eResult.SUCCESS THEN
	State:=eState.Inactive;
ELSIF transitionresult= eResult.FAILURE THEN
	State:=eState.Unconfigured;
ELSIF transitionresult= eResult.ERROR THEN
	State:=eState.ErrorProcessing;
ELSE
	ADSLOGSTR(ADSLOG_MSGTYPE_WARN,'Transitionresult from onConfigure is None','');
END_IF
END_METHOD

METHOD onDeactivate : BOOL
// ---- Init ----
transitionresult:=eResult.None;



// ---- Change ----

_mode:= eMode.Manual;




// ---- Check ----
transitionresult := eResult.SUCCESS;


// ---- Change State ----
IF transitionresult= eResult.SUCCESS THEN
	State:=eState.Inactive;
ELSIF transitionresult= eResult.FAILURE THEN
	ADSLOGSTR(ADSLOG_MSGTYPE_WARN,'Transitionresult from onDeactivate is FAILURE','');
ELSIF transitionresult= eResult.ERROR THEN
	State:=eState.ErrorProcessing;
ELSE
	ADSLOGSTR(ADSLOG_MSGTYPE_WARN,'Transitionresult from onDeactivate is None','');
END_IF
END_METHOD

METHOD onError : BOOL
// ---- Init ----
transitionresult:=eResult.None;



// ---- Change ----

_mode:= eMode.Manual;




// ---- Check ----
transitionresult := eResult.SUCCESS;


// ---- Change State ----
IF transitionresult= eResult.SUCCESS THEN
	State:=eState.Unconfigured;
ELSIF transitionresult= eResult.FAILURE THEN
	State:=eState.Finalized;
ELSIF transitionresult= eResult.ERROR THEN
	ADSLOGSTR(ADSLOG_MSGTYPE_WARN,'Transitionresult from onError is Error','');
ELSE
	ADSLOGSTR(ADSLOG_MSGTYPE_WARN,'Transitionresult from onError is None','');
END_IF
END_METHOD

METHOD onShutdown : BOOL
// ---- Init ----
transitionresult:=eResult.None;



// ---- Change ----

_mode:= eMode.Manual;




// ---- Check ----
transitionresult := eResult.SUCCESS;


// ---- Change State ----
IF transitionresult= eResult.SUCCESS THEN
	State:=eState.Finalized;
ELSIF transitionresult= eResult.FAILURE THEN
	ADSLOGSTR(ADSLOG_MSGTYPE_WARN,'Transitionresult from onShutdown is FAILURE','');
ELSIF transitionresult= eResult.ERROR THEN
	State:=eState.ErrorProcessing;
ELSE
	ADSLOGSTR(ADSLOG_MSGTYPE_WARN,'Transitionresult from onShutdown is None','');
END_IF
END_METHOD

{warning 'Add property implementation'}
PROPERTY P_ActualAxisPos : stJoint6
GET
P_ActualAxisPos:= jointpos;
END_GET
END_PROPERTY

{warning 'Add property implementation'}
PROPERTY P_ActualJointVelocity : stJoint6
GET
P_ActualJointVelocity:= jointvel;
END_GET
END_PROPERTY

{warning 'Add property implementation'}
PROPERTY P_ActualTCPPos : stPose3D
GET
P_ActualTCPPos:=tcppos;
END_GET
END_PROPERTY

{warning 'Add property implementation'}
PROPERTY P_ActualTCPVelocity : stPose3D
GET
P_ActualTCPVelocity:=tcpvel;
END_GET
END_PROPERTY

{warning 'Add property implementation'}
PROPERTY P_currentFrame : stFrame
GET
P_currentFrame := currFrame;
END_GET
SET
currFrame := P_currentFrame;
END_SET
END_PROPERTY

{warning 'Add property implementation'}
PROPERTY P_currentFrameID : UINT
GET
P_currentFrameID:= currFrame.frameId;
END_GET
END_PROPERTY

{warning 'Add property implementation'}
PROPERTY P_currentTool : FB_Tool
GET
P_currentTool:= currTool;
END_GET
SET
currTool:= P_currentTool;
END_SET
END_PROPERTY

{warning 'Add property implementation'}
PROPERTY P_IsInHomePosition : BOOL
GET
END_GET
END_PROPERTY

PROPERTY P_TargetReached : BOOL
GET
END_GET
END_PROPERTY

END_FUNCTION_BLOCK

// ---- POUs/Robots/FB_UR5_1.TcPOU
FUNCTION_BLOCK FB_UR5 EXTENDS FB_ROB_MANIP IMPLEMENTS ITF_BA_6Axis, ITF_CommunicationModul
VAR_INPUT
END_VAR
VAR_OUTPUT
END_VAR
VAR
	PiNPl: Skill_PickPlace;
END_VAR

StateMachine();


//Reference to Skills
PiNPl(Rob:=ADR(THIS^));

//ComConfig

ComConfig.sIPAddress:='127.0.0.1';
ComConfig.nPort:= 5432;

METHOD Connect : BOOL
VAR_INPUT
END_VAR
END_METHOD

PROPERTY Connected : BOOL
GET
END_GET
END_PROPERTY

METHOD Disconnect : BOOL
VAR_INPUT
END_VAR
END_METHOD

{warning 'Add method implementation '}
METHOD MC_MoveAxesRelative : BOOL
VAR_INPUT
	axes	: ARRAY [1..6] OF FB_Axis;
	offsets	: ARRAY [1..6] OF REAL;
END_VAR
END_METHOD

{warning 'Add method implementation '}
METHOD MC_MoveJ : BOOL
VAR_INPUT
	target	: stTarget3D;
END_VAR
IF _state=eState.Active THEN
// 	P_TargetReached:=FALSE;
END_IF
END_METHOD

{warning 'Add method implementation '}
METHOD MC_MoveL : BOOL
VAR_INPUT
	target	: stTarget3D;
END_VAR
END_METHOD

{warning 'Add method implementation '}
METHOD MC_ReadActualVelocity : stPose
END_METHOD

{warning 'Add method implementation '}
METHOD MC_ReadAnalogInput : LREAL
VAR_INPUT
	input	: INT;
END_VAR
END_METHOD

{warning 'Add method implementation '}
METHOD MC_ReadDigitalInput : BOOL
VAR_INPUT
	input	: INT;
END_VAR
END_METHOD

{warning 'Add method implementation '}
METHOD MC_SetDigitalOutput : BOOL
VAR_INPUT
	output	: INT;
	value	: BOOL;
END_VAR
END_METHOD

{warning 'Add method implementation '}
METHOD MC_SetOperationMode : BOOL
VAR_INPUT
	mode	: eMode;
END_VAR
_mode:=mode;
END_METHOD

METHOD MC_SpeedOverride : INT
VAR_INPUT
	factor: REAL;
END_VAR
END_METHOD

METHOD onActivate : BOOL
// ---- Init ----
transitionresult:=eResult.None;



// ---- Change ----

// _mode:= eMode.Automatic;




// ---- Check ----
transitionresult := eResult.SUCCESS;


// ---- Change State ----
IF transitionresult= eResult.SUCCESS THEN
	State:=eState.Active;
ELSIF transitionresult= eResult.FAILURE THEN
	State:=eState.Inactive;
ELSIF transitionresult= eResult.ERROR THEN
	State:=eState.ErrorProcessing;
ELSE
	ADSLOGSTR(ADSLOG_MSGTYPE_WARN,'Transitionresult from onActivate is None','');
END_IF
END_METHOD

METHOD onCleanup : BOOL
// ---- Init ----
transitionresult:=eResult.None;



// ---- Change ----

_mode:= eMode.Manual;




// ---- Check ----
transitionresult := eResult.SUCCESS;


// ---- Change State ----
IF transitionresult= eResult.SUCCESS THEN
	State:=eState.Unconfigured;
ELSIF transitionresult= eResult.FAILURE THEN
	ADSLOGSTR(ADSLOG_MSGTYPE_WARN,'Transitionresult from onCleanup is FAILURE ','');
ELSIF transitionresult= eResult.ERROR THEN
	State:=eState.ErrorProcessing;
ELSE
	ADSLOGSTR(ADSLOG_MSGTYPE_WARN,'Transitionresult from onCleanup is NONE','');
END_IF
END_METHOD

METHOD onConfigure : BOOL
// ---- Init ----
transitionresult:=eResult.None;



// ---- Change ----

_mode:= eMode.Manual;




// ---- Check ----
transitionresult := eResult.SUCCESS;


// ---- Change State ----
IF transitionresult= eResult.SUCCESS THEN
	State:=eState.Inactive;
ELSIF transitionresult= eResult.FAILURE THEN
	State:=eState.Unconfigured;
ELSIF transitionresult= eResult.ERROR THEN
	State:=eState.ErrorProcessing;
ELSE
	ADSLOGSTR(ADSLOG_MSGTYPE_WARN,'Transitionresult from onConfigure is None','');
END_IF
END_METHOD

METHOD onDeactivate : BOOL
// ---- Init ----
transitionresult:=eResult.None;



// ---- Change ----

_mode:= eMode.Manual;




// ---- Check ----
transitionresult := eResult.SUCCESS;


// ---- Change State ----
IF transitionresult= eResult.SUCCESS THEN
	State:=eState.Inactive;
ELSIF transitionresult= eResult.FAILURE THEN
	ADSLOGSTR(ADSLOG_MSGTYPE_WARN,'Transitionresult from onDeactivate is FAILURE','');
ELSIF transitionresult= eResult.ERROR THEN
	State:=eState.ErrorProcessing;
ELSE
	ADSLOGSTR(ADSLOG_MSGTYPE_WARN,'Transitionresult from onDeactivate is None','');
END_IF
END_METHOD

METHOD onError : BOOL
// ---- Init ----
transitionresult:=eResult.None;



// ---- Change ----

_mode:= eMode.Manual;




// ---- Check ----
transitionresult := eResult.SUCCESS;


// ---- Change State ----
IF transitionresult= eResult.SUCCESS THEN
	State:=eState.Unconfigured;
ELSIF transitionresult= eResult.FAILURE THEN
	State:=eState.Finalized;
ELSIF transitionresult= eResult.ERROR THEN
	ADSLOGSTR(ADSLOG_MSGTYPE_WARN,'Transitionresult from onError is Error','');
ELSE
	ADSLOGSTR(ADSLOG_MSGTYPE_WARN,'Transitionresult from onError is None','');
END_IF
END_METHOD

METHOD onShutdown : BOOL
// ---- Init ----
transitionresult:=eResult.None;



// ---- Change ----

_mode:= eMode.Manual;




// ---- Check ----
transitionresult := eResult.SUCCESS;


// ---- Change State ----
IF transitionresult= eResult.SUCCESS THEN
	State:=eState.Finalized;
ELSIF transitionresult= eResult.FAILURE THEN
	ADSLOGSTR(ADSLOG_MSGTYPE_WARN,'Transitionresult from onShutdown is FAILURE','');
ELSIF transitionresult= eResult.ERROR THEN
	State:=eState.ErrorProcessing;
ELSE
	ADSLOGSTR(ADSLOG_MSGTYPE_WARN,'Transitionresult from onShutdown is None','');
END_IF
END_METHOD

METHOD ResetConnection : BOOL
VAR_INPUT
END_VAR
END_METHOD

END_FUNCTION_BLOCK

// ---- POUs/Skills/Skill_PickPlace.TcPOU
FUNCTION_BLOCK Skill_PickPlace EXTENDS FB_Skill
VAR_INPUT
	Rob: POINTER TO FB_ROB_MANIP;
	sPickReference: STRING;
END_VAR
VAR_OUTPUT
	
END_VAR
VAR
	
END_VAR

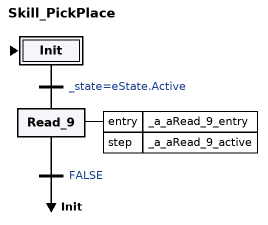
INITIAL_STEP Init:
END_STEP
TRANSITION FROM Init TO Read_9
    := _state=eState.Active;
END_TRANSITION
STEP Read_9:
    _a_aRead_9_entry(P1);  // entry action
    _a_aRead_9_active(N);  // step action
END_STEP
TRANSITION FROM Read_9 TO Init
    := FALSE;
END_TRANSITION

ACTION _a_aRead_9_active:

END_ACTION

ACTION _a_aRead_9_entry:
Rob^.MC_ReadDigitalInput(input:=8);
END_ACTION

END_FUNCTION_BLOCK

// ---- POUs/Skills/FB_SkillHandler_1.TcPOU
FUNCTION_BLOCK FB_SkillHandler
VAR_INPUT
END_VAR
VAR_OUTPUT
END_VAR
VAR
	activSkill: POINTER TO FB_SKILL;
	_finished: BOOL;
END_VAR

IF activSkill^.bDone THEN
	_finished:=True;
END_IF

METHOD AbortActifSkill : BOOL
VAR_INPUT
END_VAR
activSkill^.M_Stop();
END_METHOD

PROPERTY ActiveSkillFinished : BOOL
GET
ActiveSkillFinished := _finished;
END_GET
END_PROPERTY

METHOD CallSkill : BOOL
VAR_INPUT
	pSkill : POINTER TO FB_SKILL;
END_VAR
activSkill:= pSkill;

//TODO Checks

pSkill^.M_Start();
END_METHOD

PROPERTY GetActivSkill : POINTER TO FB_SKILL
GET
GetActivSkill := activSkill;
END_GET
END_PROPERTY

END_FUNCTION_BLOCK

// ---- POUs/Skills/FB_Skill_1.TcPOU
FUNCTION_BLOCK FB_Skill_1 EXTENDS FB_Base IMPLEMENTS  ITF_1_Skill
VAR_INPUT
	SFCInit, SFCPause, SFCReset: BOOL;
END_VAR
VAR_OUTPUT
	bBusy, bDone: BOOL;
	SFCError: BOOL;
	SFCCurrentStep: STRING;
END_VAR
VAR
	SubSkillHandler : FB_SkillHandler;
END_VAR

{warning 'Add method implementation '}
METHOD M_Pause : BOOL
IF _state=eState.Active THEN
	SFCPause:=TRUE;
END_IF
END_METHOD

{warning 'Add method implementation '}
METHOD M_Restart : BOOL //Stay activ, but restart
SFCReset:=True;
END_METHOD

{warning 'Add method implementation '}
METHOD M_Resume : BOOL
SFCPause:=False;
END_METHOD

{warning 'Add method implementation '}
METHOD M_Start : BOOL
Activate();
END_METHOD

{warning 'Add method implementation '}
METHOD M_Stop : BOOL
IF _state=eState.Active THEN
	SFCPause:=TRUE;
	super^.Deactivate();
END_IF
END_METHOD

METHOD onActivate : BOOL
// ---- Init ----
transitionresult:=eResult.None;



// ---- Change ----




// ---- Check ----
transitionresult := eResult.SUCCESS;


// ---- Change State ----
IF transitionresult= eResult.SUCCESS THEN
	State:=eState.Active;
ELSIF transitionresult= eResult.FAILURE THEN
	State:=eState.Inactive;
ELSIF transitionresult= eResult.ERROR THEN
	State:=eState.ErrorProcessing;
ELSE
	ADSLOGSTR(ADSLOG_MSGTYPE_WARN,'Transitionresult from onActivate is None','');
END_IF
END_METHOD

METHOD onCleanup : BOOL
// ---- Init ----
transitionresult:=eResult.None;



// ---- Change ----



// ---- Check ----
transitionresult := eResult.SUCCESS;


// ---- Change State ----
IF transitionresult= eResult.SUCCESS THEN
	State:=eState.Unconfigured;
ELSIF transitionresult= eResult.FAILURE THEN
	ADSLOGSTR(ADSLOG_MSGTYPE_WARN,'Transitionresult from onCleanup is FAILURE ','');
ELSIF transitionresult= eResult.ERROR THEN
	State:=eState.ErrorProcessing;
ELSE
	ADSLOGSTR(ADSLOG_MSGTYPE_WARN,'Transitionresult from onCleanup is NONE','');
END_IF
END_METHOD

METHOD onConfigure : BOOL
// ---- Init ----
transitionresult:=eResult.None;



// ---- Change ----


// ---- Check ----
transitionresult := eResult.SUCCESS;


// ---- Change State ----
IF transitionresult= eResult.SUCCESS THEN
	State:=eState.Inactive;
ELSIF transitionresult= eResult.FAILURE THEN
	State:=eState.Unconfigured;
ELSIF transitionresult= eResult.ERROR THEN
	State:=eState.ErrorProcessing;
ELSE
	ADSLOGSTR(ADSLOG_MSGTYPE_WARN,'Transitionresult from onConfigure is None','');
END_IF
END_METHOD

METHOD onDeactivate : BOOL
// ---- Init ----
transitionresult:=eResult.None;



// ---- Change ----
 //Stopping SFC



// ---- Check ----
transitionresult := eResult.SUCCESS;


// ---- Change State ----
IF transitionresult= eResult.SUCCESS THEN
	State:=eState.Inactive;
ELSIF transitionresult= eResult.FAILURE THEN
	ADSLOGSTR(ADSLOG_MSGTYPE_WARN,'Transitionresult from onDeactivate is FAILURE','');
ELSIF transitionresult= eResult.ERROR THEN
	State:=eState.ErrorProcessing;
ELSE
	ADSLOGSTR(ADSLOG_MSGTYPE_WARN,'Transitionresult from onDeactivate is None','');
END_IF
END_METHOD

METHOD onError : BOOL
// ---- Init ----
transitionresult:=eResult.None;



// ---- Change ----





// ---- Check ----
transitionresult := eResult.SUCCESS;


// ---- Change State ----
IF transitionresult= eResult.SUCCESS THEN
	State:=eState.Unconfigured;
ELSIF transitionresult= eResult.FAILURE THEN
	State:=eState.Finalized;
ELSIF transitionresult= eResult.ERROR THEN
	ADSLOGSTR(ADSLOG_MSGTYPE_WARN,'Transitionresult from onError is Error','');
ELSE
	ADSLOGSTR(ADSLOG_MSGTYPE_WARN,'Transitionresult from onError is None','');
END_IF
END_METHOD

METHOD onShutdown : BOOL
// ---- Init ----
transitionresult:=eResult.None;



// ---- Change ----




// ---- Check ----
transitionresult := eResult.SUCCESS;


// ---- Change State ----
IF transitionresult= eResult.SUCCESS THEN
	State:=eState.Finalized;
ELSIF transitionresult= eResult.FAILURE THEN
	ADSLOGSTR(ADSLOG_MSGTYPE_WARN,'Transitionresult from onShutdown is FAILURE','');
ELSIF transitionresult= eResult.ERROR THEN
	State:=eState.ErrorProcessing;
ELSE
	ADSLOGSTR(ADSLOG_MSGTYPE_WARN,'Transitionresult from onShutdown is None','');
END_IF
END_METHOD

{warning 'Add property implementation'}
PROPERTY P_Busy : BOOL
GET
IF _state=eState.Active THEN
	P_Busy:=TRUE;
ELSE
	P_Busy:=FALSE;
END_IF
END_GET
END_PROPERTY

{warning 'Add property implementation'}
PROPERTY P_Done : BOOL
GET
P_Done:=bDone;
END_GET
END_PROPERTY

END_FUNCTION_BLOCK

// ---- POUs/Skills/Skill_LoadDeliverReturn.TcPOU
FUNCTION_BLOCK Skill_LoadDeliverReturn EXTENDS FB_Skill
VAR_INPUT
	Rob: POINTER TO FB_ROB_AMR;
	sPickReference: STRING;
END_VAR
VAR_OUTPUT
	
END_VAR
VAR
	
	ActiveBAFinished: BOOL;
END_VAR

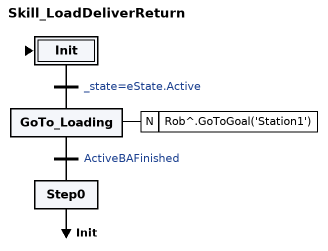
INITIAL_STEP Init:
END_STEP
TRANSITION FROM Init TO GoTo_Loading
    := _state=eState.Active;
END_TRANSITION
STEP GoTo_Loading:
    Rob^.GoToGoal('Station1')(N);
END_STEP
TRANSITION FROM GoTo_Loading TO Step0
    := ActiveBAFinished;
END_TRANSITION
STEP Step0:
END_STEP
// no transition between Step0 and Init

END_FUNCTION_BLOCK

// ---- POUs/Test.TcPOU
FUNCTION_BLOCK Test
VAR_INPUT
END_VAR
VAR_OUTPUT
END_VAR
VAR
END_VAR

METHOD Wait1S : BOOL
VAR_INPUT
END_VAR
END_METHOD

END_FUNCTION_BLOCK
